LIN {X 0,Y 249.471,Z 292.033,A -85,B 0,C 180,E1 -19088.099,E2 -19088.099} C_VEL
LIN {X 0,Y 249.243,Z 292.063,A -85,B 0,C 180,E1 -19091.385,E2 -19091.385} C_VEL
LIN {X 0,Y 249.233,Z 292.064,A -85,B 0,C 180,E1 -19096.38,E2 -19096.38} C_VEL
LIN {X 0,Y 249.075,Z 292.084,A -85,B 0,C 180,E1 -19101.52,E2 -19101.52} C_VEL
LIN {X 0,Y 249.108,Z 292.08,A -85,B 0,C 180,E1 -19105.477,E2 -19105.477} C_VEL
LIN {X 0,Y 249.043,Z 292.087,A -85,B 0,C 180,E1 -19109.572,E2 -19109.572} C_VEL
LIN {X 0,Y 248.346,Z 292.177,A -85,B 0,C 180,E1 -19110.921,E2 -19110.921} C_VEL
LIN {X 0,Y 245.475,Z 292.533,A -85,B 0,C 180,E1 -19113.119,E2 -19113.119} C_VEL
LIN {X 0,Y 243.059,Z 292.835,A -85,B 0,C 180,E1 -19114.91,E2 -19114.91} C_VEL
LIN {X 0,Y 242.033,Z 292.96,A -85,B 0,C 180,E1 -19116.299,E2 -19116.299} C_VEL
LIN {X 0,Y 241.954,Z 292.965,A -85,B 0,C 180,E1 -19116.77,E2 -19116.77} C_VEL
LIN {X 0,Y 241.928,Z 292.974,A -85,B 0,C 180,E1 -19120.953,E2 -19120.953} C_VEL
LIN {X 0,Y 241.986,Z 293.122,A -85,B 0,C 180,E1 -19124.826,E2 -19124.826} C_VEL
LIN {X 0,Y 245.244,Z 306.398,A -85,B 0,C 180,E1 -19129.049,E2 -19129.049} C_VEL
LIN {X 0,Y 245.535,Z 307.451,A -85,B 0,C 180,E1 -19129.318,E2 -19129.318} C_VEL
LIN {X 0,Y 258.623,Z 343.04,A -85,B 0,C 180,E1 -19132.403,E2 -19132.403} C_VEL
LIN {X 0,Y 260.766,Z 349.359,A -85,B 0,C 180,E1 -19132.902,E2 -19132.902} C_VEL
LIN {X 0,Y 263.208,Z 370.68,A -85,B 0,C 180,E1 -19134.126,E2 -19134.126} C_VEL
LIN {X 0,Y 255.946,Z 475.253,A -85,B 0,C 180,E1 -19138.613,E2 -19138.613} C_VEL
LIN {X 0,Y 254.356,Z 491.269,A -85,B 0,C 180,E1 -19139.606,E2 -19139.606} C_VEL
LIN {X 0,Y 252.419,Z 507.536,A -85,B 0,C 180,E1 -19140.957,E2 -19140.957} C_VEL
LIN {X 0,Y 250.356,Z 523.247,A -85,B 0,C 180,E1 -19142.636,E2 -19142.636} C_VEL
LIN {X 0,Y 248.189,Z 538.255,A -85,B 0,C 180,E1 -19144.643,E2 -19144.643} C_VEL
LIN {X 0,Y 246.113,Z 551.832,A -85,B 0,C 180,E1 -19146.883,E2 -19146.883} C_VEL
LIN {X 0,Y 244.552,Z 562.301,A -85,B 0,C 180,E1 -19148.95,E2 -19148.95} C_VEL
LIN {X 0,Y 243.07,Z 573.02,A -85,B 0,C 180,E1 -19151.458,E2 -19151.458} C_VEL
LIN {X 0,Y 241.842,Z 583.648,A -85,B 0,C 180,E1 -19154.455,E2 -19154.455} C_VEL
LIN {X 0,Y 240.981,Z 592.114,A -85,B 0,C 180,E1 -19157.368,E2 -19157.368} C_VEL
LIN {X 0,Y 240.616,Z 598.213,A -85,B 0,C 180,E1 -19159.909,E2 -19159.909} C_VEL
LIN {X 0,Y 240.531,Z 603.304,A -85,B 0,C 180,E1 -19162.447,E2 -19162.447} C_VEL
LIN {X 0,Y 240.455,Z 607.393,A -85,B 0,C 180,E1 -19164.972,E2 -19164.972} C_VEL
LIN {X 0,Y 240.557,Z 611.483,A -85,B 0,C 180,E1 -19168.328,E2 -19168.328} C_VEL
LIN {X 0,Y 240.593,Z 612.96,A -85,B 0,C 180,E1 -19170.002,E2 -19170.002} C_VEL
LIN {X 0,Y 240.362,Z 614.057,A -85,B 0,C 180,E1 -19171.678,E2 -19171.678} C_VEL
LIN {X 0,Y 240.044,Z 615.345,A -85,B 0,C 180,E1 -19175.459,E2 -19175.459} C_VEL
LIN {X 0,Y 239.986,Z 615.305,A -85,B 0,C 180,E1 -19178.422,E2 -19178.422} C_VEL
LIN {X 0,Y 240.478,Z 614.105,A -85,B 0,C 180,E1 -19181.807,E2 -19181.807} C_VEL
LIN {X 0,Y 241.79,Z 611.803,A -85,B 0,C 180,E1 -19185.167,E2 -19185.167} C_VEL
LIN {X 0,Y 243.891,Z 608.419,A -85,B 0,C 180,E1 -19188.482,E2 -19188.482} C_VEL
LIN {X 0,Y 246.847,Z 603.914,A -85,B 0,C 180,E1 -19191.725,E2 -19191.725} C_VEL
LIN {X 0,Y 251.642,Z 596.638,A -85,B 0,C 180,E1 -19195.653,E2 -19195.653} C_VEL
LIN {X 0,Y 255.249,Z 591.329,A -85,B 0,C 180,E1 -19197.912,E2 -19197.912} C_VEL
LIN {X 0,Y 261.608,Z 582.045,A -85,B 0,C 180,E1 -19201.143,E2 -19201.143} C_VEL
LIN {X 0,Y 269.062,Z 570.962,A -85,B 0,C 180,E1 -19204.168,E2 -19204.168} C_VEL
LIN {X 0,Y 276.626,Z 559.345,A -85,B 0,C 180,E1 -19206.66,E2 -19206.66} C_VEL
LIN {X 0,Y 283.903,Z 547.619,A -85,B 0,C 180,E1 -19208.689,E2 -19208.689} C_VEL
LIN {X 0,Y 291.346,Z 535.032,A -85,B 0,C 180,E1 -19210.415,E2 -19210.415} C_VEL
LIN {X 0,Y 299.334,Z 520.498,A -85,B 0,C 180,E1 -19212.003,E2 -19212.003} C_VEL
LIN {X 0,Y 305.927,Z 507.36,A -85,B 0,C 180,E1 -19213.115,E2 -19213.115} C_VEL
LIN {X 0,Y 313.351,Z 490.898,A -85,B 0,C 180,E1 -19214.214,E2 -19214.214} C_VEL
LIN {X 0,Y 320.433,Z 472.33,A -85,B 0,C 180,E1 -19215.159,E2 -19215.159} C_VEL
LIN {X 0,Y 322.394,Z 466.476,A -85,B 0,C 180,E1 -19215.395,E2 -19215.395} C_VEL
LIN {X 0,Y 321.993,Z 467.661,A -85,B 0,C 180,E1 -19215.696,E2 -19215.696} C_VEL
LIN {X 0,Y 316.048,Z 483.579,A -85,B 0,C 180,E1 -19216.64,E2 -19216.64} C_VEL
LIN {X 0,Y 309.726,Z 497.956,A -85,B 0,C 180,E1 -19217.76,E2 -19217.76} C_VEL
LIN {X 0,Y 302.493,Z 512.424,A -85,B 0,C 180,E1 -19219.197,E2 -19219.197} C_VEL
LIN {X 0,Y 295.181,Z 525.593,A -85,B 0,C 180,E1 -19220.879,E2 -19220.879} C_VEL
LIN {X 0,Y 287.732,Z 537.835,A -85,B 0,C 180,E1 -19222.804,E2 -19222.804} C_VEL
LIN {X 0,Y 280.816,Z 548.308,A -85,B 0,C 180,E1 -19224.856,E2 -19224.856} C_VEL
LIN {X 0,Y 273.456,Z 558.626,A -85,B 0,C 180,E1 -19227.335,E2 -19227.335} C_VEL
LIN {X 0,Y 266.928,Z 567.216,A -85,B 0,C 180,E1 -19229.982,E2 -19229.982} C_VEL
LIN {X 0,Y 261.165,Z 574.375,A -85,B 0,C 180,E1 -19232.775,E2 -19232.775} C_VEL
LIN {X 0,Y 256.074,Z 580.239,A -85,B 0,C 180,E1 -19235.689,E2 -19235.689} C_VEL
LIN {X 0,Y 251.537,Z 584.921,A -85,B 0,C 180,E1 -19238.701,E2 -19238.701} C_VEL
LIN {X 0,Y 248.05,Z 588.36,A -85,B 0,C 180,E1 -19241.839,E2 -19241.839} C_VEL
LIN {X 0,Y 245.208,Z 590.711,A -85,B 0,C 180,E1 -19245.05,E2 -19245.05} C_VEL
LIN {X 0,Y 243.186,Z 591.965,A -85,B 0,C 180,E1 -19248.327,E2 -19248.327} C_VEL
LIN {X 0,Y 241.569,Z 592.097,A -85,B 0,C 180,E1 -19251.635,E2 -19251.635} C_VEL
LIN {X 0,Y 240.677,Z 591.061,A -85,B 0,C 180,E1 -19254.973,E2 -19254.973} C_VEL
LIN {X 0,Y 240.242,Z 588.872,A -85,B 0,C 180,E1 -19258.322,E2 -19258.322} C_VEL
LIN {X 0,Y 240.107,Z 585.46,A -85,B 0,C 180,E1 -19261.676,E2 -19261.676} C_VEL
LIN {X 0,Y 240.137,Z 580.702,A -85,B 0,C 180,E1 -19265.036,E2 -19265.036} C_VEL
LIN {X 0,Y 240.498,Z 574.473,A -85,B 0,C 180,E1 -19268.4,E2 -19268.4} C_VEL
LIN {X 0,Y 241.056,Z 567.663,A -85,B 0,C 180,E1 -19271.348,E2 -19271.348} C_VEL
LIN {X 0,Y 242.08,Z 559.425,A -85,B 0,C 180,E1 -19274.285,E2 -19274.285} C_VEL
LIN {X 0,Y 243.19,Z 549.848,A -85,B 0,C 180,E1 -19277.122,E2 -19277.122} C_VEL
LIN {X 0,Y 244.711,Z 539.338,A -85,B 0,C 180,E1 -19279.72,E2 -19279.72} C_VEL
LIN {X 0,Y 246.494,Z 527.366,A -85,B 0,C 180,E1 -19282.195,E2 -19282.195} C_VEL
LIN {X 0,Y 248.317,Z 514.289,A -85,B 0,C 180,E1 -19284.45,E2 -19284.45} C_VEL
LIN {X 0,Y 250.42,Z 499.832,A -85,B 0,C 180,E1 -19286.501,E2 -19286.501} C_VEL
LIN {X 0,Y 252.301,Z 484.557,A -85,B 0,C 180,E1 -19288.263,E2 -19288.263} C_VEL
LIN {X 0,Y 253.967,Z 469.508,A -85,B 0,C 180,E1 -19289.645,E2 -19289.645} C_VEL
LIN {X 0,Y 255.476,Z 453.024,A -85,B 0,C 180,E1 -19290.82,E2 -19290.82} C_VEL
LIN {X 0,Y 256.778,Z 434.752,A -85,B 0,C 180,E1 -19291.74,E2 -19291.74} C_VEL
LIN {X 0,Y 263.19,Z 342.406,A -85,B 0,C 180,E1 -19295.61,E2 -19295.61} C_VEL
LIN {X 0,Y 247.394,Z 305.685,A -85,B 0,C 180,E1 -19298.918,E2 -19298.918} C_VEL
LIN {X 0,Y 242.129,Z 293.792,A -85,B 0,C 180,E1 -19300.101,E2 -19300.101} C_VEL
LIN {X 0,Y 241.983,Z 292.971,A -85,B 0,C 180,E1 -19300.199,E2 -19300.199} C_VEL
LIN {X 0,Y 241.931,Z 292.976,A -85,B 0,C 180,E1 -19304.2,E2 -19304.2} C_VEL
LIN {X 0,Y 241.938,Z 292.973,A -85,B 0,C 180,E1 -19308.075,E2 -19308.075} C_VEL
LIN {X 0,Y 241.989,Z 292.966,A -85,B 0,C 180,E1 -19312.416,E2 -19312.416} C_VEL
LIN {X 0,Y 241.978,Z 292.968,A -85,B 0,C 180,E1 -19316.505,E2 -19316.505} C_VEL
LIN {X 0,Y 241.975,Z 292.966,A -85,B 0,C 180,E1 -19320.61,E2 -19320.61} C_VEL
LIN {X 0,Y 242.03,Z 292.961,A -85,B 0,C 180,E1 -19324.176,E2 -19324.176} C_VEL
LIN {X 0,Y 242.019,Z 292.963,A -85,B 0,C 180,E1 -19328.313,E2 -19328.313} C_VEL
LIN {X 0,Y 242.111,Z 292.952,A -85,B 0,C 180,E1 -19333.314,E2 -19333.314} C_VEL
LIN {X 0,Y 242.178,Z 292.943,A -85,B 0,C 180,E1 -19338.277,E2 -19338.277} C_VEL
LIN {X 0,Y 242.422,Z 292.915,A -85,B 0,C 180,E1 -19341.663,E2 -19341.663} C_VEL
LIN {X 0,Y 242.251,Z 292.932,A -85,B 0,C 180,E1 -19345.005,E2 -19345.005} C_VEL
LIN {X 0,Y 242.629,Z 292.885,A -85,B 0,C 180,E1 -19348.338,E2 -19348.338} C_VEL
LIN {X 0,Y 242.629,Z 292.886,A -85,B 0,C 180,E1 -19351.658,E2 -19351.658} C_VEL
LIN {X 0,Y 242.425,Z 292.91,A -85,B 0,C 180,E1 -19356.657,E2 -19356.657} C_VEL
LIN {X 0,Y 242.306,Z 292.924,A -85,B 0,C 180,E1 -19360.02,E2 -19360.02} C_VEL
LIN {X 0,Y 242.157,Z 292.946,A -85,B 0,C 180,E1 -19365.139,E2 -19365.139} C_VEL
LIN {X 0,Y 242.063,Z 292.953,A -85,B 0,C 180,E1 -19368.622,E2 -19368.622} C_VEL
LIN {X 0,Y 242.003,Z 292.963,A -85,B 0,C 180,E1 -19372.178,E2 -19372.178} C_VEL
LIN {X 0,Y 242.056,Z 292.956,A -85,B 0,C 180,E1 -19375.836,E2 -19375.836} C_VEL
LIN {X 0,Y 241.996,Z 292.966,A -85,B 0,C 180,E1 -19379.582,E2 -19379.582} C_VEL
LIN {X 0,Y 241.979,Z 292.968,A -85,B 0,C 180,E1 -19383.49,E2 -19383.49} C_VEL
LIN {X 0,Y 241.987,Z 292.967,A -85,B 0,C 180,E1 -19387.579,E2 -19387.579} C_VEL
LIN {X 0,Y 241.926,Z 292.972,A -85,B 0,C 180,E1 -19391.921,E2 -19391.921} C_VEL
LIN {X 0,Y 241.924,Z 292.973,A -85,B 0,C 180,E1 -19396.57,E2 -19396.57} C_VEL
LIN {X 0,Y 241.943,Z 292.97,A -85,B 0,C 180,E1 -19400.28,E2 -19400.28} C_VEL
LIN {X 0,Y 241.974,Z 292.966,A -85,B 0,C 180,E1 -19404.489,E2 -19404.489} C_VEL
LIN {X 0,Y 241.962,Z 292.968,A -85,B 0,C 180,E1 -19408.48,E2 -19408.48} C_VEL
LIN {X 0,Y 241.994,Z 292.963,A -85,B 0,C 180,E1 -19412.313,E2 -19412.313} C_VEL
LIN {X 0,Y 242.028,Z 292.96,A -85,B 0,C 180,E1 -19416.015,E2 -19416.015} C_VEL
LIN {X 0,Y 242.022,Z 292.96,A -85,B 0,C 180,E1 -19419.608,E2 -19419.608} C_VEL
LIN {X 0,Y 242.151,Z 292.948,A -85,B 0,C 180,E1 -19423.279,E2 -19423.279} C_VEL
LIN {X 0,Y 242.174,Z 292.939,A -85,B 0,C 180,E1 -19428.281,E2 -19428.281} C_VEL
LIN {X 0,Y 242.414,Z 292.912,A -85,B 0,C 180,E1 -19431.667,E2 -19431.667} C_VEL
LIN {X 0,Y 242.246,Z 292.936,A -85,B 0,C 180,E1 -19435.008,E2 -19435.008} C_VEL
LIN {X 0,Y 242.625,Z 292.885,A -85,B 0,C 180,E1 -19438.341,E2 -19438.341} C_VEL
LIN {X 0,Y 242.625,Z 292.885,A -85,B 0,C 180,E1 -19441.661,E2 -19441.661} C_VEL
LIN {X 0,Y 242.422,Z 292.912,A -85,B 0,C 180,E1 -19446.66,E2 -19446.66} C_VEL
LIN {X 0,Y 242.304,Z 292.925,A -85,B 0,C 180,E1 -19450.023,E2 -19450.023} C_VEL
LIN {X 0,Y 242.157,Z 292.947,A -85,B 0,C 180,E1 -19455.143,E2 -19455.143} C_VEL
LIN {X 0,Y 242.062,Z 292.959,A -85,B 0,C 180,E1 -19458.626,E2 -19458.626} C_VEL
LIN {X 0,Y 241.997,Z 292.966,A -85,B 0,C 180,E1 -19462.183,E2 -19462.183} C_VEL
LIN {X 0,Y 242.059,Z 292.958,A -85,B 0,C 180,E1 -19465.84,E2 -19465.84} C_VEL
LIN {X 0,Y 242.023,Z 292.962,A -85,B 0,C 180,E1 -19469.582,E2 -19469.582} C_VEL
LIN {X 0,Y 241.973,Z 292.968,A -85,B 0,C 180,E1 -19473.495,E2 -19473.495} C_VEL
LIN {X 0,Y 241.954,Z 292.965,A -85,B 0,C 180,E1 -19476.77,E2 -19476.77} C_VEL
LIN {X 0,Y 241.262,Z 293.057,A -85,B 0,C 180,E1 -19478.16,E2 -19478.16} C_VEL
LIN {X 0,Y 238.301,Z 293.425,A -85,B 0,C 180,E1 -19480.425,E2 -19480.425} C_VEL
LIN {X 0,Y 235.86,Z 293.727,A -85,B 0,C 180,E1 -19482.272,E2 -19482.272} C_VEL
LIN {X 0,Y 234.923,Z 293.843,A -85,B 0,C 180,E1 -19483.708,E2 -19483.708} C_VEL
LIN {X 0,Y 234.906,Z 293.846,A -85,B 0,C 180,E1 -19484.193,E2 -19484.193} C_VEL
LIN {X 0,Y 238.061,Z 306.82,A -85,B 0,C 180,E1 -19488.475,E2 -19488.475} C_VEL
LIN {X 0,Y 251.779,Z 344.086,A -85,B 0,C 180,E1 -19491.829,E2 -19491.829} C_VEL
LIN {X 0,Y 254.286,Z 351.542,A -85,B 0,C 180,E1 -19492.432,E2 -19492.432} C_VEL
LIN {X 0,Y 256.465,Z 371.959,A -85,B 0,C 180,E1 -19493.631,E2 -19493.631} C_VEL
LIN {X 0,Y 249.049,Z 475.308,A -85,B 0,C 180,E1 -19498.236,E2 -19498.236} C_VEL
LIN {X 0,Y 247.449,Z 491.177,A -85,B 0,C 180,E1 -19499.257,E2 -19499.257} C_VEL
LIN {X 0,Y 245.48,Z 507.314,A -85,B 0,C 180,E1 -19500.644,E2 -19500.644} C_VEL
LIN {X 0,Y 243.495,Z 522.086,A -85,B 0,C 180,E1 -19502.266,E2 -19502.266} C_VEL
LIN {X 0,Y 241.306,Z 536.878,A -85,B 0,C 180,E1 -19504.283,E2 -19504.283} C_VEL
LIN {X 0,Y 239.163,Z 550.864,A -85,B 0,C 180,E1 -19506.63,E2 -19506.63} C_VEL
LIN {X 0,Y 237.259,Z 563.298,A -85,B 0,C 180,E1 -19509.181,E2 -19509.181} C_VEL
LIN {X 0,Y 235.803,Z 573.803,A -85,B 0,C 180,E1 -19511.766,E2 -19511.766} C_VEL
LIN {X 0,Y 234.669,Z 584.034,A -85,B 0,C 180,E1 -19514.811,E2 -19514.811} C_VEL
LIN {X 0,Y 233.873,Z 592.449,A -85,B 0,C 180,E1 -19517.859,E2 -19517.859} C_VEL
LIN {X 0,Y 233.529,Z 598.435,A -85,B 0,C 180,E1 -19520.475,E2 -19520.475} C_VEL
LIN {X 0,Y 233.493,Z 603.825,A -85,B 0,C 180,E1 -19523.361,E2 -19523.361} C_VEL
LIN {X 0,Y 233.399,Z 608.437,A -85,B 0,C 180,E1 -19526.55,E2 -19526.55} C_VEL
LIN {X 0,Y 233.51,Z 610.412,A -85,B 0,C 180,E1 -19528.278,E2 -19528.278} C_VEL
LIN {X 0,Y 233.579,Z 612.003,A -85,B 0,C 180,E1 -19530.002,E2 -19530.002} C_VEL
LIN {X 0,Y 233.316,Z 613.2,A -85,B 0,C 180,E1 -19531.728,E2 -19531.728} C_VEL
LIN {X 0,Y 232.98,Z 614.68,A -85,B 0,C 180,E1 -19535.449,E2 -19535.449} C_VEL
LIN {X 0,Y 232.934,Z 614.788,A -85,B 0,C 180,E1 -19538.679,E2 -19538.679} C_VEL
LIN {X 0,Y 233.467,Z 613.824,A -85,B 0,C 180,E1 -19542.167,E2 -19542.167} C_VEL
LIN {X 0,Y 234.887,Z 611.793,A -85,B 0,C 180,E1 -19545.624,E2 -19545.624} C_VEL
LIN {X 0,Y 237.113,Z 608.634,A -85,B 0,C 180,E1 -19549.031,E2 -19549.031} C_VEL
LIN {X 0,Y 240.255,Z 604.391,A -85,B 0,C 180,E1 -19552.353,E2 -19552.353} C_VEL
LIN {X 0,Y 244.203,Z 599.074,A -85,B 0,C 180,E1 -19555.577,E2 -19555.577} C_VEL
LIN {X 0,Y 247.692,Z 594.319,A -85,B 0,C 180,E1 -19557.918,E2 -19557.918} C_VEL
LIN {X 0,Y 254.219,Z 585.86,A -85,B 0,C 180,E1 -19561.223,E2 -19561.223} C_VEL
LIN {X 0,Y 261.679,Z 575.783,A -85,B 0,C 180,E1 -19564.335,E2 -19564.335} C_VEL
LIN {X 0,Y 269.264,Z 565.268,A -85,B 0,C 180,E1 -19566.895,E2 -19566.895} C_VEL
LIN {X 0,Y 277.722,Z 553.047,A -85,B 0,C 180,E1 -19569.248,E2 -19569.248} C_VEL
LIN {X 0,Y 285.828,Z 540.646,A -85,B 0,C 180,E1 -19571.129,E2 -19571.129} C_VEL
LIN {X 0,Y 294.614,Z 526.272,A -85,B 0,C 180,E1 -19572.835,E2 -19572.835} C_VEL
LIN {X 0,Y 301.989,Z 513.063,A -85,B 0,C 180,E1 -19574.05,E2 -19574.05} C_VEL
LIN {X 0,Y 310.398,Z 496.278,A -85,B 0,C 180,E1 -19575.244,E2 -19575.244} C_VEL
LIN {X 0,Y 311.954,Z 492.865,A -85,B 0,C 180,E1 -19575.438,E2 -19575.438} C_VEL
LIN {X 0,Y 312.63,Z 491.313,A -85,B 0,C 180,E1 -19575.821,E2 -19575.821} C_VEL
LIN {X 0,Y 304.858,Z 506.763,A -85,B 0,C 180,E1 -19577.15,E2 -19577.15} C_VEL
LIN {X 0,Y 297.467,Z 519.809,A -85,B 0,C 180,E1 -19578.582,E2 -19578.582} C_VEL
LIN {X 0,Y 289.388,Z 532.714,A -85,B 0,C 180,E1 -19580.393,E2 -19580.393} C_VEL
LIN {X 0,Y 281.786,Z 543.831,A -85,B 0,C 180,E1 -19582.333,E2 -19582.333} C_VEL
LIN {X 0,Y 273.714,Z 554.743,A -85,B 0,C 180,E1 -19584.709,E2 -19584.709} C_VEL
LIN {X 0,Y 266.275,Z 563.98,A -85,B 0,C 180,E1 -19587.242,E2 -19587.242} C_VEL
LIN {X 0,Y 259.516,Z 571.879,A -85,B 0,C 180,E1 -19590.022,E2 -19590.022} C_VEL
LIN {X 0,Y 253.824,Z 578.109,A -85,B 0,C 180,E1 -19592.814,E2 -19592.814} C_VEL
LIN {X 0,Y 248.587,Z 583.315,A -85,B 0,C 180,E1 -19595.798,E2 -19595.798} C_VEL
LIN {X 0,Y 245.121,Z 586.469,A -85,B 0,C 180,E1 -19598.115,E2 -19598.115} C_VEL
LIN {X 0,Y 241.423,Z 589.63,A -85,B 0,C 180,E1 -19601.323,E2 -19601.323} C_VEL
LIN {X 0,Y 238.419,Z 591.673,A -85,B 0,C 180,E1 -19604.614,E2 -19604.614} C_VEL
LIN {X 0,Y 236.267,Z 592.64,A -85,B 0,C 180,E1 -19607.981,E2 -19607.981} C_VEL
LIN {X 0,Y 234.5,Z 592.517,A -85,B 0,C 180,E1 -19611.51,E2 -19611.51} C_VEL
LIN {X 0,Y 233.615,Z 591.322,A -85,B 0,C 180,E1 -19614.821,E2 -19614.821} C_VEL
LIN {X 0,Y 233.169,Z 588.895,A -85,B 0,C 180,E1 -19618.271,E2 -19618.271} C_VEL
LIN {X 0,Y 233.012,Z 585.241,A -85,B 0,C 180,E1 -19621.727,E2 -19621.727} C_VEL
LIN {X 0,Y 233.063,Z 580.242,A -85,B 0,C 180,E1 -19625.189,E2 -19625.189} C_VEL
LIN {X 0,Y 233.457,Z 573.753,A -85,B 0,C 180,E1 -19628.656,E2 -19628.656} C_VEL
LIN {X 0,Y 234.039,Z 566.675,A -85,B 0,C 180,E1 -19631.693,E2 -19631.693} C_VEL
LIN {X 0,Y 235.137,Z 558.152,A -85,B 0,C 180,E1 -19634.716,E2 -19634.716} C_VEL
LIN {X 0,Y 236.389,Z 547.893,A -85,B 0,C 180,E1 -19637.726,E2 -19637.726} C_VEL
LIN {X 0,Y 237.919,Z 537.359,A -85,B 0,C 180,E1 -19640.308,E2 -19640.308} C_VEL
LIN {X 0,Y 239.844,Z 524.995,A -85,B 0,C 180,E1 -19642.844,E2 -19642.844} C_VEL
LIN {X 0,Y 241.761,Z 511.435,A -85,B 0,C 180,E1 -19645.158,E2 -19645.158} C_VEL
LIN {X 0,Y 243.852,Z 496.676,A -85,B 0,C 180,E1 -19647.218,E2 -19647.218} C_VEL
LIN {X 0,Y 245.794,Z 481.08,A -85,B 0,C 180,E1 -19648.965,E2 -19648.965} C_VEL
LIN {X 0,Y 247.553,Z 465.099,A -85,B 0,C 180,E1 -19650.376,E2 -19650.376} C_VEL
LIN {X 0,Y 248.997,Z 447.809,A -85,B 0,C 180,E1 -19651.535,E2 -19651.535} C_VEL
LIN {X 0,Y 251.431,Z 412.603,A -85,B 0,C 180,E1 -19653.162,E2 -19653.162} C_VEL
LIN {X 0,Y 256.429,Z 344.058,A -85,B 0,C 180,E1 -19656.119,E2 -19656.119} C_VEL
LIN {X 0,Y 241.327,Z 308.785,A -85,B 0,C 180,E1 -19659.384,E2 -19659.384} C_VEL
LIN {X 0,Y 234.952,Z 294.19,A -85,B 0,C 180,E1 -19660.864,E2 -19660.864} C_VEL
LIN {X 0,Y 234.911,Z 293.85,A -85,B 0,C 180,E1 -19660.918,E2 -19660.918} C_VEL
LIN {X 0,Y 234.895,Z 293.853,A -85,B 0,C 180,E1 -19664.102,E2 -19664.102} C_VEL
LIN {X 0,Y 234.883,Z 293.85,A -85,B 0,C 180,E1 -19668.83,E2 -19668.83} C_VEL
LIN {X 0,Y 234.918,Z 293.845,A -85,B 0,C 180,E1 -19671.076,E2 -19671.076} C_VEL
LIN {X 0,Y 234.929,Z 293.845,A -85,B 0,C 180,E1 -19675.359,E2 -19675.359} C_VEL
LIN {X 0,Y 234.897,Z 293.848,A -85,B 0,C 180,E1 -19679.425,E2 -19679.425} C_VEL
LIN {X 0,Y 234.966,Z 293.843,A -85,B 0,C 180,E1 -19683.804,E2 -19683.804} C_VEL
LIN {X 0,Y 234.965,Z 293.841,A -85,B 0,C 180,E1 -19688.963,E2 -19688.963} C_VEL
LIN {X 0,Y 235.052,Z 293.831,A -85,B 0,C 180,E1 -19693.09,E2 -19693.09} C_VEL
LIN {X 0,Y 235.108,Z 293.825,A -85,B 0,C 180,E1 -19697.919,E2 -19697.919} C_VEL
LIN {X 0,Y 235.372,Z 293.794,A -85,B 0,C 180,E1 -19701.412,E2 -19701.412} C_VEL
LIN {X 0,Y 235.398,Z 293.787,A -85,B 0,C 180,E1 -19703.139,E2 -19703.139} C_VEL
LIN {X 0,Y 235.588,Z 293.763,A -85,B 0,C 180,E1 -19708.288,E2 -19708.288} C_VEL
LIN {X 0,Y 235.588,Z 293.763,A -85,B 0,C 180,E1 -19711.707,E2 -19711.707} C_VEL
LIN {X 0,Y 235.396,Z 293.786,A -85,B 0,C 180,E1 -19716.856,E2 -19716.856} C_VEL
LIN {X 0,Y 235.23,Z 293.804,A -85,B 0,C 180,E1 -19720.324,E2 -19720.324} C_VEL
LIN {X 0,Y 235.104,Z 293.825,A -85,B 0,C 180,E1 -19725.604,E2 -19725.604} C_VEL
LIN {X 0,Y 234.999,Z 293.835,A -85,B 0,C 180,E1 -19729.204,E2 -19729.204} C_VEL
LIN {X 0,Y 234.951,Z 293.842,A -85,B 0,C 180,E1 -19732.881,E2 -19732.881} C_VEL
LIN {X 0,Y 234.957,Z 293.839,A -85,B 0,C 180,E1 -19736.656,E2 -19736.656} C_VEL
LIN {X 0,Y 234.911,Z 293.846,A -85,B 0,C 180,E1 -19740.568,E2 -19740.568} C_VEL
LIN {X 0,Y 234.949,Z 293.84,A -85,B 0,C 180,E1 -19744.632,E2 -19744.632} C_VEL
LIN {X 0,Y 234.93,Z 293.845,A -85,B 0,C 180,E1 -19748.943,E2 -19748.943} C_VEL
LIN {X 0,Y 234.877,Z 293.851,A -85,B 0,C 180,E1 -19753.485,E2 -19753.485} C_VEL
LIN {X 0,Y 234.877,Z 293.85,A -85,B 0,C 180,E1 -19756.514,E2 -19756.514} C_VEL
LIN {X 0,Y 234.905,Z 293.849,A -85,B 0,C 180,E1 -19761.078,E2 -19761.078} C_VEL
LIN {X 0,Y 234.917,Z 293.849,A -85,B 0,C 180,E1 -19765.362,E2 -19765.362} C_VEL
LIN {X 0,Y 234.919,Z 293.846,A -85,B 0,C 180,E1 -19769.432,E2 -19769.432} C_VEL
LIN {X 0,Y 234.981,Z 293.838,A -85,B 0,C 180,E1 -19773.794,E2 -19773.794} C_VEL
LIN {X 0,Y 234.985,Z 293.838,A -85,B 0,C 180,E1 -19778.969,E2 -19778.969} C_VEL
LIN {X 0,Y 235.084,Z 293.828,A -85,B 0,C 180,E1 -19783.06,E2 -19783.06} C_VEL
LIN {X 0,Y 235.134,Z 293.816,A -85,B 0,C 180,E1 -19787.925,E2 -19787.925} C_VEL
LIN {X 0,Y 235.364,Z 293.792,A -85,B 0,C 180,E1 -19791.415,E2 -19791.415} C_VEL
LIN {X 0,Y 235.39,Z 293.79,A -85,B 0,C 180,E1 -19793.142,E2 -19793.142} C_VEL
LIN {X 0,Y 235.584,Z 293.762,A -85,B 0,C 180,E1 -19798.292,E2 -19798.292} C_VEL
LIN {X 0,Y 235.584,Z 293.762,A -85,B 0,C 180,E1 -19801.711,E2 -19801.711} C_VEL
LIN {X 0,Y 235.393,Z 293.789,A -85,B 0,C 180,E1 -19806.86,E2 -19806.86} C_VEL
LIN {X 0,Y 235.228,Z 293.807,A -85,B 0,C 180,E1 -19810.328,E2 -19810.328} C_VEL
LIN {X 0,Y 235.104,Z 293.823,A -85,B 0,C 180,E1 -19815.608,E2 -19815.608} C_VEL
LIN {X 0,Y 234.998,Z 293.84,A -85,B 0,C 180,E1 -19819.208,E2 -19819.208} C_VEL
LIN {X 0,Y 234.944,Z 293.849,A -85,B 0,C 180,E1 -19822.886,E2 -19822.886} C_VEL
LIN {X 0,Y 234.961,Z 293.845,A -85,B 0,C 180,E1 -19826.66,E2 -19826.66} C_VEL
LIN {X 0,Y 234.924,Z 293.848,A -85,B 0,C 180,E1 -19830.57,E2 -19830.57} C_VEL
LIN {X 0,Y 234.923,Z 293.848,A -85,B 0,C 180,E1 -19834.64,E2 -19834.64} C_VEL
LIN {X 0,Y 234.936,Z 293.845,A -85,B 0,C 180,E1 -19838.947,E2 -19838.947} C_VEL
LIN {X 0,Y 234.885,Z 293.848,A -85,B 0,C 180,E1 -19843.488,E2 -19843.488} C_VEL
LIN {X 0,Y 234.906,Z 293.846,A -85,B 0,C 180,E1 -19844.193,E2 -19844.193} C_VEL
LIN {X 0,Y 234.529,Z 297.073,A -85,B 0,C 180,E1 -19845.175,E2 -19845.175} C_VEL
LIN {X 0,Y 231.193,Z 305.933,A -85,B 0,C 180,E1 -19847.406,E2 -19847.406} C_VEL
LIN {X 0,Y 231.341,Z 308.208,A -85,B 0,C 180,E1 -19847.796,E2 -19847.796} C_VEL
LIN {X 0,Y 231.483,Z 308.699,A -85,B 0,C 180,E1 -19847.849,E2 -19847.849} C_VEL
LIN {X 0,Y 244.35,Z 343.383,A -85,B 0,C 180,E1 -19851.089,E2 -19851.089} C_VEL
LIN {X 0,Y 247.822,Z 353.873,A -85,B 0,C 180,E1 -19851.962,E2 -19851.962} C_VEL
LIN {X 0,Y 249.807,Z 372.241,A -85,B 0,C 180,E1 -19853.084,E2 -19853.084} C_VEL
LIN {X 0,Y 242.249,Z 474.246,A -85,B 0,C 180,E1 -19857.789,E2 -19857.789} C_VEL
LIN {X 0,Y 240.547,Z 490.797,A -85,B 0,C 180,E1 -19858.887,E2 -19858.887} C_VEL
LIN {X 0,Y 238.54,Z 506.868,A -85,B 0,C 180,E1 -19860.311,E2 -19860.311} C_VEL
LIN {X 0,Y 236.421,Z 522.486,A -85,B 0,C 180,E1 -19862.086,E2 -19862.086} C_VEL
LIN {X 0,Y 234.338,Z 536.071,A -85,B 0,C 180,E1 -19864.004,E2 -19864.004} C_VEL
LIN {X 0,Y 232.207,Z 549.77,A -85,B 0,C 180,E1 -19866.361,E2 -19866.361} C_VEL
LIN {X 0,Y 230.258,Z 562.314,A -85,B 0,C 180,E1 -19868.986,E2 -19868.986} C_VEL
LIN {X 0,Y 228.788,Z 572.89,A -85,B 0,C 180,E1 -19871.65,E2 -19871.65} C_VEL
LIN {X 0,Y 227.621,Z 583.202,A -85,B 0,C 180,E1 -19874.788,E2 -19874.788} C_VEL
LIN {X 0,Y 226.832,Z 591.666,A -85,B 0,C 180,E1 -19877.931,E2 -19877.931} C_VEL
LIN {X 0,Y 226.477,Z 598.592,A -85,B 0,C 180,E1 -19881.077,E2 -19881.077} C_VEL
LIN {X 0,Y 226.458,Z 603.746,A -85,B 0,C 180,E1 -19883.998,E2 -19883.998} C_VEL
LIN {X 0,Y 226.409,Z 608.273,A -85,B 0,C 180,E1 -19887.334,E2 -19887.334} C_VEL
LIN {X 0,Y 226.563,Z 611.006,A -85,B 0,C 180,E1 -19890.002,E2 -19890.002} C_VEL
LIN {X 0,Y 225.974,Z 613.212,A -85,B 0,C 180,E1 -19893.569,E2 -19893.569} C_VEL
LIN {X 0,Y 225.935,Z 613.901,A -85,B 0,C 180,E1 -19895.488,E2 -19895.488} C_VEL
LIN {X 0,Y 225.871,Z 614.253,A -85,B 0,C 180,E1 -19898.953,E2 -19898.953} C_VEL
LIN {X 0,Y 226.468,Z 613.546,A -85,B 0,C 180,E1 -19902.549,E2 -19902.549} C_VEL
LIN {X 0,Y 228.002,Z 611.698,A -85,B 0,C 180,E1 -19906.109,E2 -19906.109} C_VEL
LIN {X 0,Y 230.366,Z 608.818,A -85,B 0,C 180,E1 -19909.611,E2 -19909.611} C_VEL
LIN {X 0,Y 233.708,Z 604.914,A -85,B 0,C 180,E1 -19913.015,E2 -19913.015} C_VEL
LIN {X 0,Y 239.022,Z 598.488,A -85,B 0,C 180,E1 -19917.115,E2 -19917.115} C_VEL
LIN {X 0,Y 242.996,Z 593.772,A -85,B 0,C 180,E1 -19919.453,E2 -19919.453} C_VEL
LIN {X 0,Y 249.94,Z 585.498,A -85,B 0,C 180,E1 -19922.773,E2 -19922.773} C_VEL
LIN {X 0,Y 257.979,Z 575.635,A -85,B 0,C 180,E1 -19925.856,E2 -19925.856} C_VEL
LIN {X 0,Y 266.026,Z 565.377,A -85,B 0,C 180,E1 -19928.379,E2 -19928.379} C_VEL
LIN {X 0,Y 274.94,Z 553.485,A -85,B 0,C 180,E1 -19930.682,E2 -19930.682} C_VEL
LIN {X 0,Y 283.489,Z 541.455,A -85,B 0,C 180,E1 -19932.499,E2 -19932.499} C_VEL
LIN {X 0,Y 291.95,Z 528.629,A -85,B 0,C 180,E1 -19934.037,E2 -19934.037} C_VEL
LIN {X 0,Y 299.4,Z 516.422,A -85,B 0,C 180,E1 -19935.195,E2 -19935.195} C_VEL
LIN {X 0,Y 303.894,Z 508.474,A -85,B 0,C 180,E1 -19935.803,E2 -19935.803} C_VEL
LIN {X 0,Y 295.567,Z 522.09,A -85,B 0,C 180,E1 -19937.337,E2 -19937.337} C_VEL
LIN {X 0,Y 287.102,Z 534.606,A -85,B 0,C 180,E1 -19939.093,E2 -19939.093} C_VEL
LIN {X 0,Y 279.089,Z 545.405,A -85,B 0,C 180,E1 -19940.982,E2 -19940.982} C_VEL
LIN {X 0,Y 270.55,Z 555.988,A -85,B 0,C 180,E1 -19943.311,E2 -19943.311} C_VEL
LIN {X 0,Y 262.644,Z 565.032,A -85,B 0,C 180,E1 -19945.809,E2 -19945.809} C_VEL
LIN {X 0,Y 255.577,Z 572.597,A -85,B 0,C 180,E1 -19948.501,E2 -19948.501} C_VEL
LIN {X 0,Y 249.254,Z 578.89,A -85,B 0,C 180,E1 -19951.357,E2 -19951.357} C_VEL
LIN {X 0,Y 243.675,Z 583.972,A -85,B 0,C 180,E1 -19954.365,E2 -19954.365} C_VEL
LIN {X 0,Y 238.721,Z 587.964,A -85,B 0,C 180,E1 -19957.496,E2 -19957.496} C_VEL
LIN {X 0,Y 234.814,Z 590.811,A -85,B 0,C 180,E1 -19960.777,E2 -19960.777} C_VEL
LIN {X 0,Y 231.648,Z 592.625,A -85,B 0,C 180,E1 -19964.153,E2 -19964.153} C_VEL
LIN {X 0,Y 229.351,Z 593.32,A -85,B 0,C 180,E1 -19967.612,E2 -19967.612} C_VEL
LIN {X 0,Y 227.43,Z 592.862,A -85,B 0,C 180,E1 -19971.45,E2 -19971.45} C_VEL
LIN {X 0,Y 226.537,Z 591.465,A -85,B 0,C 180,E1 -19974.658,E2 -19974.658} C_VEL
LIN {X 0,Y 226.099,Z 588.842,A -85,B 0,C 180,E1 -19978.217,E2 -19978.217} C_VEL
LIN {X 0,Y 225.92,Z 584.978,A -85,B 0,C 180,E1 -19981.781,E2 -19981.781} C_VEL
LIN {X 0,Y 225.997,Z 579.742,A -85,B 0,C 180,E1 -19985.352,E2 -19985.352} C_VEL
LIN {X 0,Y 226.411,Z 572.977,A -85,B 0,C 180,E1 -19988.927,E2 -19988.927} C_VEL
LIN {X 0,Y 227.023,Z 565.633,A -85,B 0,C 180,E1 -19992.06,E2 -19992.06} C_VEL
LIN {X 0,Y 228.177,Z 556.791,A -85,B 0,C 180,E1 -19995.176,E2 -19995.176} C_VEL
LIN {X 0,Y 229.442,Z 546.978,A -85,B 0,C 180,E1 -19998.06,E2 -19998.06} C_VEL
LIN {X 0,Y 231.155,Z 535.304,A -85,B 0,C 180,E1 -20000.929,E2 -20000.929} C_VEL
LIN {X 0,Y 233.145,Z 522.427,A -85,B 0,C 180,E1 -20003.54,E2 -20003.54} C_VEL
LIN {X 0,Y 235.208,Z 508.234,A -85,B 0,C 180,E1 -20005.911,E2 -20005.911} C_VEL
LIN {X 0,Y 237.174,Z 494.344,A -85,B 0,C 180,E1 -20007.819,E2 -20007.819} C_VEL
LIN {X 0,Y 239.205,Z 478.306,A -85,B 0,C 180,E1 -20009.599,E2 -20009.599} C_VEL
LIN {X 0,Y 240.998,Z 461.613,A -85,B 0,C 180,E1 -20011.049,E2 -20011.049} C_VEL
LIN {X 0,Y 242.393,Z 444.81,A -85,B 0,C 180,E1 -20012.129,E2 -20012.129} C_VEL
LIN {X 0,Y 249.659,Z 345.549,A -85,B 0,C 180,E1 -20016.652,E2 -20016.652} C_VEL
LIN {X 0,Y 234.565,Z 310.363,A -85,B 0,C 180,E1 -20020.01,E2 -20020.01} C_VEL
LIN {X 0,Y 227.938,Z 295.232,A -85,B 0,C 180,E1 -20021.619,E2 -20021.619} C_VEL
LIN {X 0,Y 227.849,Z 294.73,A -85,B 0,C 180,E1 -20021.712,E2 -20021.712} C_VEL
LIN {X 0,Y 227.834,Z 294.731,A -85,B 0,C 180,E1 -20025.19,E2 -20025.19} C_VEL
LIN {X 0,Y 227.826,Z 294.732,A -85,B 0,C 180,E1 -20029.621,E2 -20029.621} C_VEL
LIN {X 0,Y 227.88,Z 294.723,A -85,B 0,C 180,E1 -20034.126,E2 -20034.126} C_VEL
LIN {X 0,Y 227.854,Z 294.725,A -85,B 0,C 180,E1 -20038.373,E2 -20038.373} C_VEL
LIN {X 0,Y 227.853,Z 294.726,A -85,B 0,C 180,E1 -20042.438,E2 -20042.438} C_VEL
LIN {X 0,Y 227.891,Z 294.721,A -85,B 0,C 180,E1 -20046.362,E2 -20046.362} C_VEL
LIN {X 0,Y 227.91,Z 294.721,A -85,B 0,C 180,E1 -20050.169,E2 -20050.169} C_VEL
LIN {X 0,Y 228.016,Z 294.71,A -85,B 0,C 180,E1 -20053.892,E2 -20053.892} C_VEL
LIN {X 0,Y 228.063,Z 294.703,A -85,B 0,C 180,E1 -20057.54,E2 -20057.54} C_VEL
LIN {X 0,Y 228.301,Z 294.673,A -85,B 0,C 180,E1 -20061.144,E2 -20061.144} C_VEL
LIN {X 0,Y 228.349,Z 294.665,A -85,B 0,C 180,E1 -20062.926,E2 -20062.926} C_VEL
LIN {X 0,Y 228.547,Z 294.64,A -85,B 0,C 180,E1 -20068.235,E2 -20068.235} C_VEL
LIN {X 0,Y 228.547,Z 294.64,A -85,B 0,C 180,E1 -20071.76,E2 -20071.76} C_VEL
LIN {X 0,Y 228.347,Z 294.665,A -85,B 0,C 180,E1 -20077.069,E2 -20077.069} C_VEL
LIN {X 0,Y 228.151,Z 294.686,A -85,B 0,C 180,E1 -20080.648,E2 -20080.648} C_VEL
LIN {X 0,Y 228.056,Z 294.701,A -85,B 0,C 180,E1 -20084.27,E2 -20084.27} C_VEL
LIN {X 0,Y 227.994,Z 294.706,A -85,B 0,C 180,E1 -20087.951,E2 -20087.951} C_VEL
LIN {X 0,Y 227.92,Z 294.717,A -85,B 0,C 180,E1 -20092.327,E2 -20092.327} C_VEL
LIN {X 0,Y 227.931,Z 294.714,A -85,B 0,C 180,E1 -20096.601,E2 -20096.601} C_VEL
LIN {X 0,Y 227.886,Z 294.721,A -85,B 0,C 180,E1 -20100.29,E2 -20100.29} C_VEL
LIN {X 0,Y 227.878,Z 294.722,A -85,B 0,C 180,E1 -20103.717,E2 -20103.717} C_VEL
LIN {X 0,Y 227.837,Z 294.727,A -85,B 0,C 180,E1 -20108.089,E2 -20108.089} C_VEL
LIN {X 0,Y 227.8,Z 294.732,A -85,B 0,C 180,E1 -20112.741,E2 -20112.741} C_VEL
LIN {X 0,Y 227.8,Z 294.736,A -85,B 0,C 180,E1 -20117.257,E2 -20117.257} C_VEL
LIN {X 0,Y 227.831,Z 294.725,A -85,B 0,C 180,E1 -20121.909,E2 -20121.909} C_VEL
LIN {X 0,Y 227.866,Z 294.724,A -85,B 0,C 180,E1 -20126.377,E2 -20126.377} C_VEL
LIN {X 0,Y 227.906,Z 294.717,A -85,B 0,C 180,E1 -20130.438,E2 -20130.438} C_VEL
LIN {X 0,Y 227.912,Z 294.718,A -85,B 0,C 180,E1 -20134.426,E2 -20134.426} C_VEL
LIN {X 0,Y 227.935,Z 294.714,A -85,B 0,C 180,E1 -20138.286,E2 -20138.286} C_VEL
LIN {X 0,Y 228.022,Z 294.706,A -85,B 0,C 180,E1 -20142.827,E2 -20142.827} C_VEL
LIN {X 0,Y 228.082,Z 294.696,A -85,B 0,C 180,E1 -20147.545,E2 -20147.545} C_VEL
LIN {X 0,Y 228.293,Z 294.674,A -85,B 0,C 180,E1 -20151.147,E2 -20151.147} C_VEL
LIN {X 0,Y 228.341,Z 294.668,A -85,B 0,C 180,E1 -20152.93,E2 -20152.93} C_VEL
LIN {X 0,Y 228.543,Z 294.639,A -85,B 0,C 180,E1 -20158.239,E2 -20158.239} C_VEL
LIN {X 0,Y 228.543,Z 294.639,A -85,B 0,C 180,E1 -20161.764,E2 -20161.764} C_VEL
LIN {X 0,Y 228.344,Z 294.668,A -85,B 0,C 180,E1 -20167.073,E2 -20167.073} C_VEL
LIN {X 0,Y 228.153,Z 294.69,A -85,B 0,C 180,E1 -20170.652,E2 -20170.652} C_VEL
LIN {X 0,Y 228.055,Z 294.702,A -85,B 0,C 180,E1 -20174.274,E2 -20174.274} C_VEL
LIN {X 0,Y 227.994,Z 294.71,A -85,B 0,C 180,E1 -20177.955,E2 -20177.955} C_VEL
LIN {X 0,Y 227.908,Z 294.722,A -85,B 0,C 180,E1 -20182.323,E2 -20182.323} C_VEL
LIN {X 0,Y 227.935,Z 294.72,A -85,B 0,C 180,E1 -20186.605,E2 -20186.605} C_VEL
LIN {X 0,Y 227.901,Z 294.722,A -85,B 0,C 180,E1 -20190.298,E2 -20190.298} C_VEL
LIN {X 0,Y 227.87,Z 294.724,A -85,B 0,C 180,E1 -20193.723,E2 -20193.723} C_VEL
LIN {X 0,Y 227.837,Z 294.728,A -85,B 0,C 180,E1 -20198.094,E2 -20198.094} C_VEL
LIN {X 0,Y 227.807,Z 294.731,A -85,B 0,C 180,E1 -20202.745,E2 -20202.745} C_VEL
LIN {X 0,Y 227.888,Z 294.888,A -85,B 0,C 180,E1 -20203.711,E2 -20203.711} C_VEL
LIN {X 0,Y 230.803,Z 306.7,A -85,B 0,C 180,E1 -20207.657,E2 -20207.657} C_VEL
LIN {X 0,Y 231.483,Z 308.699,A -85,B 0,C 180,E1 -20207.849,E2 -20207.849} C_VEL
LIN {X 0,Y 232.114,Z 312.47,A -85,B 0,C 180,E1 -20208.136,E2 -20208.136} C_VEL
LIN {X 0,Y 231.267,Z 325.668,A -85,B 0,C 180,E1 -20208.794,E2 -20208.794} C_VEL
LIN {X 0,Y 231.995,Z 329.4,A -85,B 0,C 180,E1 -20209.083,E2 -20209.083} C_VEL
LIN {X 0,Y 241.276,Z 355.391,A -85,B 0,C 180,E1 -20211.438,E2 -20211.438} C_VEL
LIN {X 0,Y 243.139,Z 372.64,A -85,B 0,C 180,E1 -20212.524,E2 -20212.524} C_VEL
LIN {X 0,Y 235.311,Z 474.772,A -85,B 0,C 180,E1 -20217.427,E2 -20217.427} C_VEL
LIN {X 0,Y 233.512,Z 491.51,A -85,B 0,C 180,E1 -20218.6,E2 -20218.6} C_VEL
LIN {X 0,Y 231.353,Z 508.287,A -85,B 0,C 180,E1 -20220.173,E2 -20220.173} C_VEL
LIN {X 0,Y 229.352,Z 522.687,A -85,B 0,C 180,E1 -20221.895,E2 -20221.895} C_VEL
LIN {X 0,Y 227.162,Z 536.714,A -85,B 0,C 180,E1 -20223.959,E2 -20223.959} C_VEL
LIN {X 0,Y 225.081,Z 549.758,A -85,B 0,C 180,E1 -20226.299,E2 -20226.299} C_VEL
LIN {X 0,Y 223.279,Z 561.233,A -85,B 0,C 180,E1 -20228.781,E2 -20228.781} C_VEL
LIN {X 0,Y 221.781,Z 571.876,A -85,B 0,C 180,E1 -20231.528,E2 -20231.528} C_VEL
LIN {X 0,Y 220.608,Z 582.296,A -85,B 0,C 180,E1 -20234.765,E2 -20234.765} C_VEL
LIN {X 0,Y 219.788,Z 590.827,A -85,B 0,C 180,E1 -20238.007,E2 -20238.007} C_VEL
LIN {X 0,Y 219.476,Z 596.844,A -85,B 0,C 180,E1 -20240.789,E2 -20240.789} C_VEL
LIN {X 0,Y 219.469,Z 602.343,A -85,B 0,C 180,E1 -20243.862,E2 -20243.862} C_VEL
LIN {X 0,Y 219.41,Z 607.035,A -85,B 0,C 180,E1 -20247.249,E2 -20247.249} C_VEL
LIN {X 0,Y 219.544,Z 609.874,A -85,B 0,C 180,E1 -20250.003,E2 -20250.003} C_VEL
LIN {X 0,Y 219.239,Z 611.259,A -85,B 0,C 180,E1 -20251.839,E2 -20251.839} C_VEL
LIN {X 0,Y 218.89,Z 613.081,A -85,B 0,C 180,E1 -20255.53,E2 -20255.53} C_VEL
LIN {X 0,Y 218.827,Z 613.7,A -85,B 0,C 180,E1 -20259.243,E2 -20259.243} C_VEL
LIN {X 0,Y 219.486,Z 613.154,A -85,B 0,C 180,E1 -20262.955,E2 -20262.955} C_VEL
LIN {X 0,Y 221.139,Z 611.59,A -85,B 0,C 180,E1 -20266.623,E2 -20266.623} C_VEL
LIN {X 0,Y 223.653,Z 609.006,A -85,B 0,C 180,E1 -20270.224,E2 -20270.224} C_VEL
LIN {X 0,Y 228.201,Z 604.312,A -85,B 0,C 180,E1 -20274.57,E2 -20274.57} C_VEL
LIN {X 0,Y 233.995,Z 598.013,A -85,B 0,C 180,E1 -20278.724,E2 -20278.724} C_VEL
LIN {X 0,Y 241.643,Z 589.948,A -85,B 0,C 180,E1 -20282.553,E2 -20282.553} C_VEL
LIN {X 0,Y 249.628,Z 581.192,A -85,B 0,C 180,E1 -20285.748,E2 -20285.748} C_VEL
LIN {X 0,Y 257.644,Z 572.1,A -85,B 0,C 180,E1 -20288.36,E2 -20288.36} C_VEL
LIN {X 0,Y 266.499,Z 561.585,A -85,B 0,C 180,E1 -20290.747,E2 -20290.747} C_VEL
LIN {X 0,Y 274.939,Z 550.998,A -85,B 0,C 180,E1 -20292.642,E2 -20292.642} C_VEL
LIN {X 0,Y 284.032,Z 538.905,A -85,B 0,C 180,E1 -20294.35,E2 -20294.35} C_VEL
LIN {X 0,Y 292.661,Z 526.48,A -85,B 0,C 180,E1 -20295.734,E2 -20295.734} C_VEL
LIN {X 0,Y 293.672,Z 524.992,A -85,B 0,C 180,E1 -20295.887,E2 -20295.887} C_VEL
LIN {X 0,Y 293.883,Z 524.636,A -85,B 0,C 180,E1 -20296.09,E2 -20296.09} C_VEL
LIN {X 0,Y 285.037,Z 536.658,A -85,B 0,C 180,E1 -20297.786,E2 -20297.786} C_VEL
LIN {X 0,Y 276.626,Z 547.127,A -85,B 0,C 180,E1 -20299.619,E2 -20299.619} C_VEL
LIN {X 0,Y 267.659,Z 557.397,A -85,B 0,C 180,E1 -20301.898,E2 -20301.898} C_VEL
LIN {X 0,Y 259.266,Z 566.22,A -85,B 0,C 180,E1 -20304.351,E2 -20304.351} C_VEL
LIN {X 0,Y 251.695,Z 573.61,A -85,B 0,C 180,E1 -20307.009,E2 -20307.009} C_VEL
LIN {X 0,Y 244.944,Z 579.763,A -85,B 0,C 180,E1 -20309.859,E2 -20309.859} C_VEL
LIN {X 0,Y 237.526,Z 585.806,A -85,B 0,C 180,E1 -20313.651,E2 -20313.651} C_VEL
LIN {X 0,Y 232.341,Z 589.489,A -85,B 0,C 180,E1 -20316.843,E2 -20316.843} C_VEL
LIN {X 0,Y 228.227,Z 591.989,A -85,B 0,C 180,E1 -20320.199,E2 -20320.199} C_VEL
LIN {X 0,Y 224.865,Z 593.478,A -85,B 0,C 180,E1 -20323.662,E2 -20323.662} C_VEL
LIN {X 0,Y 222.441,Z 593.936,A -85,B 0,C 180,E1 -20327.221,E2 -20327.221} C_VEL
LIN {X 0,Y 220.548,Z 593.337,A -85,B 0,C 180,E1 -20330.831,E2 -20330.831} C_VEL
LIN {X 0,Y 219.465,Z 591.582,A -85,B 0,C 180,E1 -20334.486,E2 -20334.486} C_VEL
LIN {X 0,Y 219.03,Z 588.696,A -85,B 0,C 180,E1 -20338.16,E2 -20338.16} C_VEL
LIN {X 0,Y 218.832,Z 584.575,A -85,B 0,C 180,E1 -20341.839,E2 -20341.839} C_VEL
LIN {X 0,Y 218.932,Z 579.081,A -85,B 0,C 180,E1 -20345.525,E2 -20345.525} C_VEL
LIN {X 0,Y 219.363,Z 572.033,A -85,B 0,C 180,E1 -20349.216,E2 -20349.216} C_VEL
LIN {X 0,Y 220.036,Z 564.42,A -85,B 0,C 180,E1 -20352.449,E2 -20352.449} C_VEL
LIN {X 0,Y 221.234,Z 555.258,A -85,B 0,C 180,E1 -20355.664,E2 -20355.664} C_VEL
LIN {X 0,Y 222.691,Z 544.595,A -85,B 0,C 180,E1 -20358.771,E2 -20358.771} C_VEL
LIN {X 0,Y 224.439,Z 532.961,A -85,B 0,C 180,E1 -20361.587,E2 -20361.587} C_VEL
LIN {X 0,Y 226.324,Z 520.784,A -85,B 0,C 180,E1 -20364.05,E2 -20364.05} C_VEL
LIN {X 0,Y 228.447,Z 506.647,A -85,B 0,C 180,E1 -20366.427,E2 -20366.427} C_VEL
LIN {X 0,Y 230.565,Z 491.991,A -85,B 0,C 180,E1 -20368.441,E2 -20368.441} C_VEL
LIN {X 0,Y 232.534,Z 476.433,A -85,B 0,C 180,E1 -20370.161,E2 -20370.161} C_VEL
LIN {X 0,Y 234.266,Z 459.597,A -85,B 0,C 180,E1 -20371.603,E2 -20371.603} C_VEL
LIN {X 0,Y 235.815,Z 442.215,A -85,B 0,C 180,E1 -20372.694,E2 -20372.694} C_VEL
LIN {X 0,Y 242.919,Z 347.235,A -85,B 0,C 180,E1 -20377.174,E2 -20377.174} C_VEL
LIN {X 0,Y 227.43,Z 311.058,A -85,B 0,C 180,E1 -20380.754,E2 -20380.754} C_VEL
LIN {X 0,Y 220.89,Z 296.316,A -85,B 0,C 180,E1 -20382.386,E2 -20382.386} C_VEL
LIN {X 0,Y 220.787,Z 295.61,A -85,B 0,C 180,E1 -20382.515,E2 -20382.515} C_VEL
LIN {X 0,Y 220.766,Z 295.61,A -85,B 0,C 180,E1 -20387.068,E2 -20387.068} C_VEL
LIN {X 0,Y 220.806,Z 295.603,A -85,B 0,C 180,E1 -20390.46,E2 -20390.46} C_VEL
LIN {X 0,Y 220.8,Z 295.604,A -85,B 0,C 180,E1 -20395.042,E2 -20395.042} C_VEL
LIN {X 0,Y 220.832,Z 295.6,A -85,B 0,C 180,E1 -20399.387,E2 -20399.387} C_VEL
LIN {X 0,Y 220.873,Z 295.598,A -85,B 0,C 180,E1 -20403.544,E2 -20403.544} C_VEL
LIN {X 0,Y 220.863,Z 295.599,A -85,B 0,C 180,E1 -20407.549,E2 -20407.549} C_VEL
LIN {X 0,Y 220.924,Z 295.59,A -85,B 0,C 180,E1 -20412.615,E2 -20412.615} C_VEL
LIN {X 0,Y 220.999,Z 295.581,A -85,B 0,C 180,E1 -20417.135,E2 -20417.135} C_VEL
LIN {X 0,Y 221.231,Z 295.553,A -85,B 0,C 180,E1 -20420.858,E2 -20420.858} C_VEL
LIN {X 0,Y 221.284,Z 295.545,A -85,B 0,C 180,E1 -20422.699,E2 -20422.699} C_VEL
LIN {X 0,Y 221.505,Z 295.517,A -85,B 0,C 180,E1 -20428.179,E2 -20428.179} C_VEL
LIN {X 0,Y 221.505,Z 295.516,A -85,B 0,C 180,E1 -20431.816,E2 -20431.816} C_VEL
LIN {X 0,Y 221.298,Z 295.545,A -85,B 0,C 180,E1 -20437.296,E2 -20437.296} C_VEL
LIN {X 0,Y 221.098,Z 295.565,A -85,B 0,C 180,E1 -20440.992,E2 -20440.992} C_VEL
LIN {X 0,Y 221.007,Z 295.578,A -85,B 0,C 180,E1 -20446.628,E2 -20446.628} C_VEL
LIN {X 0,Y 220.883,Z 295.593,A -85,B 0,C 180,E1 -20450.484,E2 -20450.484} C_VEL
LIN {X 0,Y 220.857,Z 295.597,A -85,B 0,C 180,E1 -20454.433,E2 -20454.433} C_VEL
LIN {X 0,Y 220.816,Z 295.601,A -85,B 0,C 180,E1 -20458.513,E2 -20458.513} C_VEL
LIN {X 0,Y 220.811,Z 295.603,A -85,B 0,C 180,E1 -20462.754,E2 -20462.754} C_VEL
LIN {X 0,Y 220.827,Z 295.602,A -85,B 0,C 180,E1 -20467.287,E2 -20467.287} C_VEL
LIN {X 0,Y 220.758,Z 295.609,A -85,B 0,C 180,E1 -20471.951,E2 -20471.951} C_VEL
LIN {X 0,Y 220.763,Z 295.61,A -85,B 0,C 180,E1 -20475.546,E2 -20475.546} C_VEL
LIN {X 0,Y 220.794,Z 295.604,A -85,B 0,C 180,E1 -20480.463,E2 -20480.463} C_VEL
LIN {X 0,Y 220.788,Z 295.607,A -85,B 0,C 180,E1 -20485.045,E2 -20485.045} C_VEL
LIN {X 0,Y 220.855,Z 295.597,A -85,B 0,C 180,E1 -20489.395,E2 -20489.395} C_VEL
LIN {X 0,Y 220.882,Z 295.595,A -85,B 0,C 180,E1 -20493.55,E2 -20493.55} C_VEL
LIN {X 0,Y 220.853,Z 295.597,A -85,B 0,C 180,E1 -20497.552,E2 -20497.552} C_VEL
LIN {X 0,Y 220.972,Z 295.583,A -85,B 0,C 180,E1 -20502.572,E2 -20502.572} C_VEL
LIN {X 0,Y 221.014,Z 295.578,A -85,B 0,C 180,E1 -20507.14,E2 -20507.14} C_VEL
LIN {X 0,Y 221.224,Z 295.553,A -85,B 0,C 180,E1 -20510.862,E2 -20510.862} C_VEL
LIN {X 0,Y 221.276,Z 295.547,A -85,B 0,C 180,E1 -20512.703,E2 -20512.703} C_VEL
LIN {X 0,Y 221.501,Z 295.516,A -85,B 0,C 180,E1 -20518.183,E2 -20518.183} C_VEL
LIN {X 0,Y 221.501,Z 295.516,A -85,B 0,C 180,E1 -20521.82,E2 -20521.82} C_VEL
LIN {X 0,Y 221.279,Z 295.546,A -85,B 0,C 180,E1 -20527.3,E2 -20527.3} C_VEL
LIN {X 0,Y 221.102,Z 295.57,A -85,B 0,C 180,E1 -20530.996,E2 -20530.996} C_VEL
LIN {X 0,Y 221.007,Z 295.581,A -85,B 0,C 180,E1 -20536.632,E2 -20536.632} C_VEL
LIN {X 0,Y 220.875,Z 295.599,A -85,B 0,C 180,E1 -20540.489,E2 -20540.489} C_VEL
LIN {X 0,Y 220.854,Z 295.601,A -85,B 0,C 180,E1 -20544.438,E2 -20544.438} C_VEL
LIN {X 0,Y 220.829,Z 295.605,A -85,B 0,C 180,E1 -20548.516,E2 -20548.516} C_VEL
LIN {X 0,Y 220.811,Z 295.607,A -85,B 0,C 180,E1 -20552.758,E2 -20552.758} C_VEL
LIN {X 0,Y 220.804,Z 295.605,A -85,B 0,C 180,E1 -20557.281,E2 -20557.281} C_VEL
LIN {X 0,Y 220.765,Z 295.607,A -85,B 0,C 180,E1 -20561.955,E2 -20561.955} C_VEL
LIN {X 0,Y 220.815,Z 295.723,A -85,B 0,C 180,E1 -20563.124,E2 -20563.124} C_VEL
LIN {X 0,Y 223.394,Z 306.266,A -85,B 0,C 180,E1 -20566.762,E2 -20566.762} C_VEL
LIN {X 0,Y 231.995,Z 329.4,A -85,B 0,C 180,E1 -20569.083,E2 -20569.083} C_VEL
LIN {X 0,Y 233.452,Z 334.808,A -85,B 0,C 180,E1 -20569.537,E2 -20569.537} C_VEL
LIN {X 0,Y 234.302,Z 344.316,A -85,B 0,C 180,E1 -20570.155,E2 -20570.155} C_VEL
LIN {X 0,Y 234.436,Z 352.106,A -85,B 0,C 180,E1 -20570.604,E2 -20570.604} C_VEL
LIN {X 0,Y 234.974,Z 359.83,A -85,B 0,C 180,E1 -20571.087,E2 -20571.087} C_VEL
LIN {X 0,Y 236.377,Z 373.799,A -85,B 0,C 180,E1 -20571.988,E2 -20571.988} C_VEL
LIN {X 0,Y 228.461,Z 473.89,A -85,B 0,C 180,E1 -20576.974,E2 -20576.974} C_VEL
LIN {X 0,Y 226.629,Z 490.769,A -85,B 0,C 180,E1 -20578.188,E2 -20578.188} C_VEL
LIN {X 0,Y 224.439,Z 507.523,A -85,B 0,C 180,E1 -20579.806,E2 -20579.806} C_VEL
LIN {X 0,Y 222.279,Z 522.754,A -85,B 0,C 180,E1 -20581.691,E2 -20581.691} C_VEL
LIN {X 0,Y 219.992,Z 537.392,A -85,B 0,C 180,E1 -20583.946,E2 -20583.946} C_VEL
LIN {X 0,Y 217.769,Z 550.683,A -85,B 0,C 180,E1 -20586.464,E2 -20586.464} C_VEL
LIN {X 0,Y 216.016,Z 561.979,A -85,B 0,C 180,E1 -20589.033,E2 -20589.033} C_VEL
LIN {X 0,Y 214.535,Z 572.214,A -85,B 0,C 180,E1 -20591.811,E2 -20591.811} C_VEL
LIN {X 0,Y 213.576,Z 581.291,A -85,B 0,C 180,E1 -20594.74,E2 -20594.74} C_VEL
LIN {X 0,Y 212.772,Z 589.904,A -85,B 0,C 180,E1 -20598.089,E2 -20598.089} C_VEL
LIN {X 0,Y 212.469,Z 596.916,A -85,B 0,C 180,E1 -20601.442,E2 -20601.442} C_VEL
LIN {X 0,Y 212.464,Z 601.791,A -85,B 0,C 180,E1 -20604.308,E2 -20604.308} C_VEL
LIN {X 0,Y 212.459,Z 606.794,A -85,B 0,C 180,E1 -20608.107,E2 -20608.107} C_VEL
LIN {X 0,Y 212.524,Z 608.716,A -85,B 0,C 180,E1 -20610.003,E2 -20610.003} C_VEL
LIN {X 0,Y 212.229,Z 610.227,A -85,B 0,C 180,E1 -20611.9,E2 -20611.9} C_VEL
LIN {X 0,Y 211.826,Z 612.241,A -85,B 0,C 180,E1 -20615.715,E2 -20615.715} C_VEL
LIN {X 0,Y 211.8,Z 613.025,A -85,B 0,C 180,E1 -20619.553,E2 -20619.553} C_VEL
LIN {X 0,Y 212.523,Z 612.758,A -85,B 0,C 180,E1 -20623.387,E2 -20623.387} C_VEL
LIN {X 0,Y 214.278,Z 611.445,A -85,B 0,C 180,E1 -20627.171,E2 -20627.171} C_VEL
LIN {X 0,Y 216.96,Z 609.093,A -85,B 0,C 180,E1 -20630.877,E2 -20630.877} C_VEL
LIN {X 0,Y 221.756,Z 604.781,A -85,B 0,C 180,E1 -20635.334,E2 -20635.334} C_VEL
LIN {X 0,Y 227.86,Z 598.934,A -85,B 0,C 180,E1 -20639.573,E2 -20639.573} C_VEL
LIN {X 0,Y 235.624,Z 591.625,A -85,B 0,C 180,E1 -20643.366,E2 -20643.366} C_VEL
LIN {X 0,Y 243.15,Z 584.206,A -85,B 0,C 180,E1 -20646.339,E2 -20646.339} C_VEL
LIN {X 0,Y 252.389,Z 574.701,A -85,B 0,C 180,E1 -20649.311,E2 -20649.311} C_VEL
LIN {X 0,Y 261.533,Z 564.858,A -85,B 0,C 180,E1 -20651.692,E2 -20651.692} C_VEL
LIN {X 0,Y 270.184,Z 555.054,A -85,B 0,C 180,E1 -20653.578,E2 -20653.578} C_VEL
LIN {X 0,Y 280.348,Z 542.751,A -85,B 0,C 180,E1 -20655.417,E2 -20655.417} C_VEL
LIN {X 0,Y 283.617,Z 538.535,A -85,B 0,C 180,E1 -20655.943,E2 -20655.943} C_VEL
LIN {X 0,Y 284.49,Z 537.383,A -85,B 0,C 180,E1 -20656.234,E2 -20656.234} C_VEL
LIN {X 0,Y 276.105,Z 547.179,A -85,B 0,C 180,E1 -20657.879,E2 -20657.879} C_VEL
LIN {X 0,Y 266.133,Z 557.831,A -85,B 0,C 180,E1 -20660.178,E2 -20660.178} C_VEL
LIN {X 0,Y 258.299,Z 565.557,A -85,B 0,C 180,E1 -20662.25,E2 -20662.25} C_VEL
LIN {X 0,Y 250.461,Z 572.671,A -85,B 0,C 180,E1 -20664.661,E2 -20664.661} C_VEL
LIN {X 0,Y 242.576,Z 579.319,A -85,B 0,C 180,E1 -20667.588,E2 -20667.588} C_VEL
LIN {X 0,Y 235.908,Z 584.451,A -85,B 0,C 180,E1 -20670.556,E2 -20670.556} C_VEL
LIN {X 0,Y 228.488,Z 589.405,A -85,B 0,C 180,E1 -20674.492,E2 -20674.492} C_VEL
LIN {X 0,Y 223.713,Z 592.135,A -85,B 0,C 180,E1 -20677.852,E2 -20677.852} C_VEL
LIN {X 0,Y 219.711,Z 593.887,A -85,B 0,C 180,E1 -20681.343,E2 -20681.343} C_VEL
LIN {X 0,Y 216.724,Z 594.537,A -85,B 0,C 180,E1 -20684.963,E2 -20684.963} C_VEL
LIN {X 0,Y 214.456,Z 594.174,A -85,B 0,C 180,E1 -20688.659,E2 -20688.659} C_VEL
LIN {X 0,Y 212.89,Z 592.763,A -85,B 0,C 180,E1 -20692.411,E2 -20692.411} C_VEL
LIN {X 0,Y 212.151,Z 590.242,A -85,B 0,C 180,E1 -20696.2,E2 -20696.2} C_VEL
LIN {X 0,Y 211.817,Z 586.489,A -85,B 0,C 180,E1 -20699.999,E2 -20699.999} C_VEL
LIN {X 0,Y 211.758,Z 581.431,A -85,B 0,C 180,E1 -20703.804,E2 -20703.804} C_VEL
LIN {X 0,Y 212.06,Z 574.877,A -85,B 0,C 180,E1 -20707.632,E2 -20707.632} C_VEL
LIN {X 0,Y 212.594,Z 567.805,A -85,B 0,C 180,E1 -20710.956,E2 -20710.956} C_VEL
LIN {X 0,Y 213.588,Z 559.248,A -85,B 0,C 180,E1 -20714.286,E2 -20714.286} C_VEL
LIN {X 0,Y 214.929,Z 548.965,A -85,B 0,C 180,E1 -20717.603,E2 -20717.603} C_VEL
LIN {X 0,Y 216.494,Z 538.479,A -85,B 0,C 180,E1 -20720.422,E2 -20720.422} C_VEL
LIN {X 0,Y 218.475,Z 526.127,A -85,B 0,C 180,E1 -20723.206,E2 -20723.206} C_VEL
LIN {X 0,Y 220.494,Z 512.619,A -85,B 0,C 180,E1 -20725.738,E2 -20725.738} C_VEL
LIN {X 0,Y 222.689,Z 498.514,A -85,B 0,C 180,E1 -20727.908,E2 -20727.908} C_VEL
LIN {X 0,Y 224.666,Z 483.628,A -85,B 0,C 180,E1 -20729.773,E2 -20729.773} C_VEL
LIN {X 0,Y 226.508,Z 468.207,A -85,B 0,C 180,E1 -20731.311,E2 -20731.311} C_VEL
LIN {X 0,Y 228.164,Z 451.131,A -85,B 0,C 180,E1 -20732.617,E2 -20732.617} C_VEL
LIN {X 0,Y 229.889,Z 428.495,A -85,B 0,C 180,E1 -20733.853,E2 -20733.853} C_VEL
LIN {X 0,Y 236.201,Z 348.958,A -85,B 0,C 180,E1 -20737.708,E2 -20737.708} C_VEL
LIN {X 0,Y 220.833,Z 312.991,A -85,B 0,C 180,E1 -20741.389,E2 -20741.389} C_VEL
LIN {X 0,Y 213.875,Z 297.334,A -85,B 0,C 180,E1 -20743.187,E2 -20743.187} C_VEL
LIN {X 0,Y 213.728,Z 296.488,A -85,B 0,C 180,E1 -20743.317,E2 -20743.317} C_VEL
LIN {X 0,Y 213.706,Z 296.491,A -85,B 0,C 180,E1 -20746.341,E2 -20746.341} C_VEL
LIN {X 0,Y 213.717,Z 296.488,A -85,B 0,C 180,E1 -20749.14,E2 -20749.14} C_VEL
LIN {X 0,Y 213.743,Z 296.486,A -85,B 0,C 180,E1 -20753.709,E2 -20753.709} C_VEL
LIN {X 0,Y 213.757,Z 296.481,A -85,B 0,C 180,E1 -20758.258,E2 -20758.258} C_VEL
LIN {X 0,Y 213.786,Z 296.478,A -85,B 0,C 180,E1 -20762.595,E2 -20762.595} C_VEL
LIN {X 0,Y 213.807,Z 296.476,A -85,B 0,C 180,E1 -20766.977,E2 -20766.977} C_VEL
LIN {X 0,Y 213.887,Z 296.467,A -85,B 0,C 180,E1 -20772.796,E2 -20772.796} C_VEL
LIN {X 0,Y 213.937,Z 296.46,A -85,B 0,C 180,E1 -20776.703,E2 -20776.703} C_VEL
LIN {X 0,Y 214.163,Z 296.433,A -85,B 0,C 180,E1 -20780.554,E2 -20780.554} C_VEL
LIN {X 0,Y 214.222,Z 296.424,A -85,B 0,C 180,E1 -20782.457,E2 -20782.457} C_VEL
LIN {X 0,Y 214.438,Z 296.398,A -85,B 0,C 180,E1 -20788.119,E2 -20788.119} C_VEL
LIN {X 0,Y 214.544,Z 296.383,A -85,B 0,C 180,E1 -20789.997,E2 -20789.997} C_VEL
LIN {X 0,Y 214.438,Z 296.396,A -85,B 0,C 180,E1 -20791.876,E2 -20791.876} C_VEL
LIN {X 0,Y 214.233,Z 296.425,A -85,B 0,C 180,E1 -20797.538,E2 -20797.538} C_VEL
LIN {X 0,Y 214.015,Z 296.449,A -85,B 0,C 180,E1 -20801.361,E2 -20801.361} C_VEL
LIN {X 0,Y 213.925,Z 296.463,A -85,B 0,C 180,E1 -20805.235,E2 -20805.235} C_VEL
LIN {X 0,Y 213.83,Z 296.471,A -85,B 0,C 180,E1 -20809.185,E2 -20809.185} C_VEL
LIN {X 0,Y 213.837,Z 296.474,A -85,B 0,C 180,E1 -20813.225,E2 -20813.225} C_VEL
LIN {X 0,Y 213.818,Z 296.474,A -85,B 0,C 180,E1 -20817.448,E2 -20817.448} C_VEL
LIN {X 0,Y 213.759,Z 296.483,A -85,B 0,C 180,E1 -20821.736,E2 -20821.736} C_VEL
LIN {X 0,Y 213.737,Z 296.482,A -85,B 0,C 180,E1 -20826.286,E2 -20826.286} C_VEL
LIN {X 0,Y 213.7,Z 296.491,A -85,B 0,C 180,E1 -20831.124,E2 -20831.124} C_VEL
LIN {X 0,Y 213.695,Z 296.488,A -85,B 0,C 180,E1 -20833.677,E2 -20833.677} C_VEL
LIN {X 0,Y 213.695,Z 296.489,A -85,B 0,C 180,E1 -20836.343,E2 -20836.343} C_VEL
LIN {X 0,Y 213.705,Z 296.491,A -85,B 0,C 180,E1 -20839.142,E2 -20839.142} C_VEL
LIN {X 0,Y 213.731,Z 296.485,A -85,B 0,C 180,E1 -20843.711,E2 -20843.711} C_VEL
LIN {X 0,Y 213.782,Z 296.479,A -85,B 0,C 180,E1 -20848.725,E2 -20848.725} C_VEL
LIN {X 0,Y 213.814,Z 296.474,A -85,B 0,C 180,E1 -20852.603,E2 -20852.603} C_VEL
LIN {X 0,Y 213.807,Z 296.478,A -85,B 0,C 180,E1 -20856.974,E2 -20856.974} C_VEL
LIN {X 0,Y 213.931,Z 296.461,A -85,B 0,C 180,E1 -20862.804,E2 -20862.804} C_VEL
LIN {X 0,Y 213.968,Z 296.455,A -85,B 0,C 180,E1 -20866.709,E2 -20866.709} C_VEL
LIN {X 0,Y 214.155,Z 296.432,A -85,B 0,C 180,E1 -20870.557,E2 -20870.557} C_VEL
LIN {X 0,Y 214.215,Z 296.425,A -85,B 0,C 180,E1 -20872.461,E2 -20872.461} C_VEL
LIN {X 0,Y 214.434,Z 296.397,A -85,B 0,C 180,E1 -20878.123,E2 -20878.123} C_VEL
LIN {X 0,Y 214.539,Z 296.384,A -85,B 0,C 180,E1 -20880.001,E2 -20880.001} C_VEL
LIN {X 0,Y 214.434,Z 296.397,A -85,B 0,C 180,E1 -20881.88,E2 -20881.88} C_VEL
LIN {X 0,Y 214.217,Z 296.425,A -85,B 0,C 180,E1 -20887.542,E2 -20887.542} C_VEL
LIN {X 0,Y 214.035,Z 296.449,A -85,B 0,C 180,E1 -20891.364,E2 -20891.364} C_VEL
LIN {X 0,Y 213.924,Z 296.464,A -85,B 0,C 180,E1 -20895.239,E2 -20895.239} C_VEL
LIN {X 0,Y 213.827,Z 296.477,A -85,B 0,C 180,E1 -20899.19,E2 -20899.19} C_VEL
LIN {X 0,Y 213.803,Z 296.48,A -85,B 0,C 180,E1 -20903.233,E2 -20903.233} C_VEL
LIN {X 0,Y 213.822,Z 296.477,A -85,B 0,C 180,E1 -20907.452,E2 -20907.452} C_VEL
LIN {X 0,Y 213.77,Z 296.481,A -85,B 0,C 180,E1 -20911.739,E2 -20911.739} C_VEL
LIN {X 0,Y 213.737,Z 296.485,A -85,B 0,C 180,E1 -20916.291,E2 -20916.291} C_VEL
LIN {X 0,Y 213.707,Z 296.487,A -85,B 0,C 180,E1 -20921.128,E2 -20921.128} C_VEL
LIN {X 0,Y 213.747,Z 296.628,A -85,B 0,C 180,E1 -20922.541,E2 -20922.541} C_VEL
LIN {X 0,Y 216.044,Z 305.859,A -85,B 0,C 180,E1 -20925.847,E2 -20925.847} C_VEL
LIN {X 0,Y 229.452,Z 342.299,A -85,B 0,C 180,E1 -20929.55,E2 -20929.55} C_VEL
LIN {X 0,Y 234.796,Z 357.67,A -85,B 0,C 180,E1 -20930.95,E2 -20930.95} C_VEL
LIN {X 0,Y 234.974,Z 359.83,A -85,B 0,C 180,E1 -20931.087,E2 -20931.087} C_VEL
LIN {X 0,Y 235.097,Z 363.646,A -85,B 0,C 180,E1 -20931.31,E2 -20931.31} C_VEL
LIN {X 0,Y 234.605,Z 367.494,A -85,B 0,C 180,E1 -20931.478,E2 -20931.478} C_VEL
LIN {X 0,Y 232.501,Z 375.112,A -85,B 0,C 180,E1 -20931.713,E2 -20931.713} C_VEL
LIN {X 0,Y 228.945,Z 386.647,A -85,B 0,C 180,E1 -20932.049,E2 -20932.049} C_VEL
LIN {X 0,Y 228.326,Z 390.572,A -85,B 0,C 180,E1 -20932.218,E2 -20932.218} C_VEL
LIN {X 0,Y 221.569,Z 473.673,A -85,B 0,C 180,E1 -20936.559,E2 -20936.559} C_VEL
LIN {X 0,Y 219.651,Z 491.023,A -85,B 0,C 180,E1 -20937.867,E2 -20937.867} C_VEL
LIN {X 0,Y 217.414,Z 507.593,A -85,B 0,C 180,E1 -20939.532,E2 -20939.532} C_VEL
LIN {X 0,Y 215.206,Z 522.693,A -85,B 0,C 180,E1 -20941.475,E2 -20941.475} C_VEL
LIN {X 0,Y 212.886,Z 537.191,A -85,B 0,C 180,E1 -20943.8,E2 -20943.8} C_VEL
LIN {X 0,Y 210.674,Z 550.418,A -85,B 0,C 180,E1 -20946.405,E2 -20946.405} C_VEL
LIN {X 0,Y 208.797,Z 562.584,A -85,B 0,C 180,E1 -20949.306,E2 -20949.306} C_VEL
LIN {X 0,Y 207.306,Z 572.829,A -85,B 0,C 180,E1 -20952.238,E2 -20952.238} C_VEL
LIN {X 0,Y 206.419,Z 581.576,A -85,B 0,C 180,E1 -20955.208,E2 -20955.208} C_VEL
LIN {X 0,Y 205.711,Z 590.032,A -85,B 0,C 180,E1 -20958.674,E2 -20958.674} C_VEL
LIN {X 0,Y 205.471,Z 596.923,A -85,B 0,C 180,E1 -20962.139,E2 -20962.139} C_VEL
LIN {X 0,Y 205.447,Z 601.637,A -85,B 0,C 180,E1 -20965.097,E2 -20965.097} C_VEL
LIN {X 0,Y 205.475,Z 606.494,A -85,B 0,C 180,E1 -20969.023,E2 -20969.023} C_VEL
LIN {X 0,Y 205.514,Z 607.486,A -85,B 0,C 180,E1 -20970.003,E2 -20970.003} C_VEL
LIN {X 0,Y 205.215,Z 609.08,A -85,B 0,C 180,E1 -20971.965,E2 -20971.965} C_VEL
LIN {X 0,Y 204.797,Z 611.292,A -85,B 0,C 180,E1 -20975.912,E2 -20975.912} C_VEL
LIN {X 0,Y 204.758,Z 612.34,A -85,B 0,C 180,E1 -20979.884,E2 -20979.884} C_VEL
LIN {X 0,Y 205.576,Z 612.289,A -85,B 0,C 180,E1 -20983.848,E2 -20983.848} C_VEL
LIN {X 0,Y 208.31,Z 610.621,A -85,B 0,C 180,E1 -20989.146,E2 -20989.146} C_VEL
LIN {X 0,Y 212.144,Z 607.789,A -85,B 0,C 180,E1 -20993.427,E2 -20993.427} C_VEL
LIN {X 0,Y 217.749,Z 603.273,A -85,B 0,C 180,E1 -20997.907,E2 -20997.907} C_VEL
LIN {X 0,Y 223.314,Z 598.578,A -85,B 0,C 180,E1 -21001.286,E2 -21001.286} C_VEL
LIN {X 0,Y 231.891,Z 591.273,A -85,B 0,C 180,E1 -21005.161,E2 -21005.161} C_VEL
LIN {X 0,Y 241.769,Z 582.359,A -85,B 0,C 180,E1 -21008.683,E2 -21008.683} C_VEL
LIN {X 0,Y 251.806,Z 572.82,A -85,B 0,C 180,E1 -21011.522,E2 -21011.522} C_VEL
LIN {X 0,Y 262.871,Z 561.665,A -85,B 0,C 180,E1 -21014.04,E2 -21014.04} C_VEL
LIN {X 0,Y 273.554,Z 550.115,A -85,B 0,C 180,E1 -21016.004,E2 -21016.004} C_VEL
LIN {X 0,Y 274.948,Z 548.545,A -85,B 0,C 180,E1 -21016.357,E2 -21016.357} C_VEL
LIN {X 0,Y 264.934,Z 558.514,A -85,B 0,C 180,E1 -21018.456,E2 -21018.456} C_VEL
LIN {X 0,Y 255.496,Z 567.111,A -85,B 0,C 180,E1 -21020.752,E2 -21020.752} C_VEL
LIN {X 0,Y 246.748,Z 574.405,A -85,B 0,C 180,E1 -21023.263,E2 -21023.263} C_VEL
LIN {X 0,Y 238.833,Z 580.45,A -85,B 0,C 180,E1 -21026.005,E2 -21026.005} C_VEL
LIN {X 0,Y 230.015,Z 586.534,A -85,B 0,C 180,E1 -21029.724,E2 -21029.724} C_VEL
LIN {X 0,Y 222.266,Z 591.009,A -85,B 0,C 180,E1 -21033.724,E2 -21033.724} C_VEL
LIN {X 0,Y 217.257,Z 593.384,A -85,B 0,C 180,E1 -21037.157,E2 -21037.157} C_VEL
LIN {X 0,Y 213.043,Z 594.779,A -85,B 0,C 180,E1 -21040.737,E2 -21040.737} C_VEL
LIN {X 0,Y 209.91,Z 595.184,A -85,B 0,C 180,E1 -21044.462,E2 -21044.462} C_VEL
LIN {X 0,Y 207.508,Z 594.557,A -85,B 0,C 180,E1 -21048.274,E2 -21048.274} C_VEL
LIN {X 0,Y 205.857,Z 592.848,A -85,B 0,C 180,E1 -21052.15,E2 -21052.15} C_VEL
LIN {X 0,Y 205.076,Z 590.055,A -85,B 0,C 180,E1 -21056.068,E2 -21056.068} C_VEL
LIN {X 0,Y 204.749,Z 586.081,A -85,B 0,C 180,E1 -21059.998,E2 -21059.998} C_VEL
LIN {X 0,Y 204.685,Z 580.771,A -85,B 0,C 180,E1 -21063.936,E2 -21063.936} C_VEL
LIN {X 0,Y 205.008,Z 573.96,A -85,B 0,C 180,E1 -21067.88,E2 -21067.88} C_VEL
LIN {X 0,Y 205.587,Z 566.583,A -85,B 0,C 180,E1 -21071.334,E2 -21071.334} C_VEL
LIN {X 0,Y 206.692,Z 557.721,A -85,B 0,C 180,E1 -21074.773,E2 -21074.773} C_VEL
LIN {X 0,Y 208.068,Z 547.23,A -85,B 0,C 180,E1 -21078.14,E2 -21078.14} C_VEL
LIN {X 0,Y 209.93,Z 535.131,A -85,B 0,C 180,E1 -21081.349,E2 -21081.349} C_VEL
LIN {X 0,Y 212.041,Z 522.078,A -85,B 0,C 180,E1 -21084.213,E2 -21084.213} C_VEL
LIN {X 0,Y 214.238,Z 507.674,A -85,B 0,C 180,E1 -21086.81,E2 -21086.81} C_VEL
LIN {X 0,Y 216.375,Z 493.453,A -85,B 0,C 180,E1 -21088.906,E2 -21088.906} C_VEL
LIN {X 0,Y 218.539,Z 477.287,A -85,B 0,C 180,E1 -21090.831,E2 -21090.831} C_VEL
LIN {X 0,Y 220.385,Z 460.786,A -85,B 0,C 180,E1 -21092.352,E2 -21092.352} C_VEL
LIN {X 0,Y 221.918,Z 443.777,A -85,B 0,C 180,E1 -21093.518,E2 -21093.518} C_VEL
LIN {X 0,Y 229.465,Z 350.682,A -85,B 0,C 180,E1 -21098.257,E2 -21098.257} C_VEL
LIN {X 0,Y 214.632,Z 315.789,A -85,B 0,C 180,E1 -21101.931,E2 -21101.931} C_VEL
LIN {X 0,Y 206.727,Z 297.839,A -85,B 0,C 180,E1 -21104.071,E2 -21104.071} C_VEL
LIN {X 0,Y 206.639,Z 297.373,A -85,B 0,C 180,E1 -21104.139,E2 -21104.139} C_VEL
LIN {X 0,Y 206.642,Z 297.369,A -85,B 0,C 180,E1 -21108.434,E2 -21108.434} C_VEL
LIN {X 0,Y 206.68,Z 297.366,A -85,B 0,C 180,E1 -21112.257,E2 -21112.257} C_VEL
LIN {X 0,Y 206.694,Z 297.364,A -85,B 0,C 180,E1 -21117.039,E2 -21117.039} C_VEL
LIN {X 0,Y 206.707,Z 297.361,A -85,B 0,C 180,E1 -21122.124,E2 -21122.124} C_VEL
LIN {X 0,Y 206.742,Z 297.355,A -85,B 0,C 180,E1 -21126.607,E2 -21126.607} C_VEL
LIN {X 0,Y 206.821,Z 297.348,A -85,B 0,C 180,E1 -21132.189,E2 -21132.189} C_VEL
LIN {X 0,Y 206.876,Z 297.341,A -85,B 0,C 180,E1 -21136.24,E2 -21136.24} C_VEL
LIN {X 0,Y 207.101,Z 297.314,A -85,B 0,C 180,E1 -21140.228,E2 -21140.228} C_VEL
LIN {X 0,Y 207.163,Z 297.304,A -85,B 0,C 180,E1 -21142.198,E2 -21142.198} C_VEL
LIN {X 0,Y 207.375,Z 297.278,A -85,B 0,C 180,E1 -21148.055,E2 -21148.055} C_VEL
LIN {X 0,Y 207.508,Z 297.259,A -85,B 0,C 180,E1 -21149.997,E2 -21149.997} C_VEL
LIN {X 0,Y 207.375,Z 297.275,A -85,B 0,C 180,E1 -21151.939,E2 -21151.939} C_VEL
LIN {X 0,Y 207.17,Z 297.303,A -85,B 0,C 180,E1 -21157.796,E2 -21157.796} C_VEL
LIN {X 0,Y 206.935,Z 297.333,A -85,B 0,C 180,E1 -21161.755,E2 -21161.755} C_VEL
LIN {X 0,Y 206.858,Z 297.342,A -85,B 0,C 180,E1 -21165.768,E2 -21165.768} C_VEL
LIN {X 0,Y 206.774,Z 297.351,A -85,B 0,C 180,E1 -21169.867,E2 -21169.867} C_VEL
LIN {X 0,Y 206.753,Z 297.354,A -85,B 0,C 180,E1 -21174.07,E2 -21174.07} C_VEL
LIN {X 0,Y 206.726,Z 297.356,A -85,B 0,C 180,E1 -21178.418,E2 -21178.418} C_VEL
LIN {X 0,Y 206.694,Z 297.363,A -85,B 0,C 180,E1 -21182.955,E2 -21182.955} C_VEL
LIN {X 0,Y 206.711,Z 297.359,A -85,B 0,C 180,E1 -21185.319,E2 -21185.319} C_VEL
LIN {X 0,Y 206.651,Z 297.367,A -85,B 0,C 180,E1 -21190.249,E2 -21190.249} C_VEL
LIN {X 0,Y 206.622,Z 297.372,A -85,B 0,C 180,E1 -21195.581,E2 -21195.581} C_VEL
LIN {X 0,Y 206.648,Z 297.367,A -85,B 0,C 180,E1 -21199.748,E2 -21199.748} C_VEL
LIN {X 0,Y 206.686,Z 297.362,A -85,B 0,C 180,E1 -21204.688,E2 -21204.688} C_VEL
LIN {X 0,Y 206.711,Z 297.359,A -85,B 0,C 180,E1 -21209.339,E2 -21209.339} C_VEL
LIN {X 0,Y 206.719,Z 297.359,A -85,B 0,C 180,E1 -21213.772,E2 -21213.772} C_VEL
LIN {X 0,Y 206.726,Z 297.355,A -85,B 0,C 180,E1 -21218.042,E2 -21218.042} C_VEL
LIN {X 0,Y 206.86,Z 297.34,A -85,B 0,C 180,E1 -21222.197,E2 -21222.197} C_VEL
LIN {X 0,Y 206.902,Z 297.334,A -85,B 0,C 180,E1 -21226.246,E2 -21226.246} C_VEL
LIN {X 0,Y 207.094,Z 297.311,A -85,B 0,C 180,E1 -21230.232,E2 -21230.232} C_VEL
LIN {X 0,Y 207.155,Z 297.304,A -85,B 0,C 180,E1 -21232.202,E2 -21232.202} C_VEL
LIN {X 0,Y 207.371,Z 297.277,A -85,B 0,C 180,E1 -21238.059,E2 -21238.059} C_VEL
LIN {X 0,Y 207.504,Z 297.26,A -85,B 0,C 180,E1 -21240.002,E2 -21240.002} C_VEL
LIN {X 0,Y 207.371,Z 297.277,A -85,B 0,C 180,E1 -21241.944,E2 -21241.944} C_VEL
LIN {X 0,Y 207.158,Z 297.304,A -85,B 0,C 180,E1 -21247.801,E2 -21247.801} C_VEL
LIN {X 0,Y 206.972,Z 297.328,A -85,B 0,C 180,E1 -21251.757,E2 -21251.757} C_VEL
LIN {X 0,Y 206.858,Z 297.342,A -85,B 0,C 180,E1 -21255.773,E2 -21255.773} C_VEL
LIN {X 0,Y 206.754,Z 297.357,A -85,B 0,C 180,E1 -21259.873,E2 -21259.873} C_VEL
LIN {X 0,Y 206.739,Z 297.359,A -85,B 0,C 180,E1 -21264.077,E2 -21264.077} C_VEL
LIN {X 0,Y 206.737,Z 297.36,A -85,B 0,C 180,E1 -21268.421,E2 -21268.421} C_VEL
LIN {X 0,Y 206.696,Z 297.365,A -85,B 0,C 180,E1 -21272.96,E2 -21272.96} C_VEL
LIN {X 0,Y 206.674,Z 297.365,A -85,B 0,C 180,E1 -21277.743,E2 -21277.743} C_VEL
LIN {X 0,Y 206.681,Z 297.525,A -85,B 0,C 180,E1 -21281.945,E2 -21281.945} C_VEL
LIN {X 0,Y 208.645,Z 305.506,A -85,B 0,C 180,E1 -21284.89,E2 -21284.89} C_VEL
LIN {X 0,Y 220.109,Z 336.47,A -85,B 0,C 180,E1 -21288.213,E2 -21288.213} C_VEL
LIN {X 0,Y 228.245,Z 359.523,A -85,B 0,C 180,E1 -21290.423,E2 -21290.423} C_VEL
LIN {X 0,Y 229.682,Z 374.179,A -85,B 0,C 180,E1 -21291.404,E2 -21291.404} C_VEL
LIN {X 0,Y 228.326,Z 390.572,A -85,B 0,C 180,E1 -21292.218,E2 -21292.218} C_VEL
LIN {X 0,Y 227.153,Z 396.303,A -85,B 0,C 180,E1 -21292.446,E2 -21292.446} C_VEL
LIN {X 0,Y 220.012,Z 414.729,A -85,B 0,C 180,E1 -21292.938,E2 -21292.938} C_VEL
LIN {X 0,Y 218.987,Z 420.451,A -85,B 0,C 180,E1 -21293.201,E2 -21293.201} C_VEL
LIN {X 0,Y 214.613,Z 474.032,A -85,B 0,C 180,E1 -21296.175,E2 -21296.175} C_VEL
LIN {X 0,Y 212.662,Z 491.06,A -85,B 0,C 180,E1 -21297.522,E2 -21297.522} C_VEL
LIN {X 0,Y 210.558,Z 506.466,A -85,B 0,C 180,E1 -21299.127,E2 -21299.127} C_VEL
LIN {X 0,Y 208.315,Z 521.44,A -85,B 0,C 180,E1 -21301.1,E2 -21301.1} C_VEL
LIN {X 0,Y 206.004,Z 535.63,A -85,B 0,C 180,E1 -21303.417,E2 -21303.417} C_VEL
LIN {X 0,Y 203.771,Z 548.988,A -85,B 0,C 180,E1 -21306.096,E2 -21306.096} C_VEL
LIN {X 0,Y 201.836,Z 561.263,A -85,B 0,C 180,E1 -21309.093,E2 -21309.093} C_VEL
LIN {X 0,Y 200.331,Z 571.626,A -85,B 0,C 180,E1 -21312.127,E2 -21312.127} C_VEL
LIN {X 0,Y 199.419,Z 580.458,A -85,B 0,C 180,E1 -21315.199,E2 -21315.199} C_VEL
LIN {X 0,Y 198.7,Z 588.985,A -85,B 0,C 180,E1 -21318.785,E2 -21318.785} C_VEL
LIN {X 0,Y 198.481,Z 596.184,A -85,B 0,C 180,E1 -21322.509,E2 -21322.509} C_VEL
LIN {X 0,Y 198.444,Z 601.423,A -85,B 0,C 180,E1 -21325.941,E2 -21325.941} C_VEL
LIN {X 0,Y 198.502,Z 605.151,A -85,B 0,C 180,E1 -21328.988,E2 -21328.988} C_VEL
LIN {X 0,Y 198.526,Z 606.143,A -85,B 0,C 180,E1 -21330.003,E2 -21330.003} C_VEL
LIN {X 0,Y 198.212,Z 607.857,A -85,B 0,C 180,E1 -21332.035,E2 -21332.035} C_VEL
LIN {X 0,Y 197.765,Z 610.327,A -85,B 0,C 180,E1 -21336.123,E2 -21336.123} C_VEL
LIN {X 0,Y 197.734,Z 611.551,A -85,B 0,C 180,E1 -21340.239,E2 -21340.239} C_VEL
LIN {X 0,Y 198.647,Z 611.744,A -85,B 0,C 180,E1 -21344.342,E2 -21344.342} C_VEL
LIN {X 0,Y 200.632,Z 610.973,A -85,B 0,C 180,E1 -21348.379,E2 -21348.379} C_VEL
LIN {X 0,Y 203.669,Z 609.172,A -85,B 0,C 180,E1 -21352.31,E2 -21352.31} C_VEL
LIN {X 0,Y 207.814,Z 606.493,A -85,B 0,C 180,E1 -21356.084,E2 -21356.084} C_VEL
LIN {X 0,Y 214.254,Z 601.836,A -85,B 0,C 180,E1 -21360.562,E2 -21360.562} C_VEL
LIN {X 0,Y 220.807,Z 596.991,A -85,B 0,C 180,E1 -21363.851,E2 -21363.851} C_VEL
LIN {X 0,Y 228.188,Z 591.239,A -85,B 0,C 180,E1 -21366.914,E2 -21366.914} C_VEL
LIN {X 0,Y 238.692,Z 582.613,A -85,B 0,C 180,E1 -21370.376,E2 -21370.376} C_VEL
LIN {X 0,Y 249.274,Z 573.413,A -85,B 0,C 180,E1 -21373.136,E2 -21373.136} C_VEL
LIN {X 0,Y 261.094,Z 562.414,A -85,B 0,C 180,E1 -21375.618,E2 -21375.618} C_VEL
LIN {X 0,Y 263.542,Z 560.056,A -85,B 0,C 180,E1 -21376.059,E2 -21376.059} C_VEL
LIN {X 0,Y 265.367,Z 558.242,A -85,B 0,C 180,E1 -21376.481,E2 -21376.481} C_VEL
LIN {X 0,Y 255.351,Z 566.825,A -85,B 0,C 180,E1 -21378.657,E2 -21378.657} C_VEL
LIN {X 0,Y 245.952,Z 574.157,A -85,B 0,C 180,E1 -21381.049,E2 -21381.049} C_VEL
LIN {X 0,Y 237.326,Z 580.309,A -85,B 0,C 180,E1 -21383.681,E2 -21383.681} C_VEL
LIN {X 0,Y 227.68,Z 586.472,A -85,B 0,C 180,E1 -21387.302,E2 -21387.302} C_VEL
LIN {X 0,Y 222.472,Z 589.437,A -85,B 0,C 180,E1 -21389.638,E2 -21389.638} C_VEL
LIN {X 0,Y 216.068,Z 592.504,A -85,B 0,C 180,E1 -21392.91,E2 -21392.91} C_VEL
LIN {X 0,Y 210.835,Z 594.559,A -85,B 0,C 180,E1 -21396.42,E2 -21396.42} C_VEL
LIN {X 0,Y 206.404,Z 595.676,A -85,B 0,C 180,E1 -21400.091,E2 -21400.091} C_VEL
LIN {X 0,Y 203.089,Z 595.732,A -85,B 0,C 180,E1 -21403.927,E2 -21403.927} C_VEL
LIN {X 0,Y 200.56,Z 594.829,A -85,B 0,C 180,E1 -21407.861,E2 -21407.861} C_VEL
LIN {X 0,Y 198.829,Z 592.903,A -85,B 0,C 180,E1 -21411.87,E2 -21411.87} C_VEL
LIN {X 0,Y 198.003,Z 589.825,A -85,B 0,C 180,E1 -21415.928,E2 -21415.928} C_VEL
LIN {X 0,Y 197.683,Z 585.567,A -85,B 0,C 180,E1 -21419.998,E2 -21419.998} C_VEL
LIN {X 0,Y 197.617,Z 579.966,A -85,B 0,C 180,E1 -21424.077,E2 -21424.077} C_VEL
LIN {X 0,Y 197.923,Z 573.55,A -85,B 0,C 180,E1 -21427.797,E2 -21427.797} C_VEL
LIN {X 0,Y 198.486,Z 566.37,A -85,B 0,C 180,E1 -21431.228,E2 -21431.228} C_VEL
LIN {X 0,Y 199.601,Z 557.396,A -85,B 0,C 180,E1 -21434.788,E2 -21434.788} C_VEL
LIN {X 0,Y 200.789,Z 548.246,A -85,B 0,C 180,E1 -21437.833,E2 -21437.833} C_VEL
LIN {X 0,Y 202.424,Z 537.538,A -85,B 0,C 180,E1 -21440.845,E2 -21440.845} C_VEL
LIN {X 0,Y 204.502,Z 524.907,A -85,B 0,C 180,E1 -21443.814,E2 -21443.814} C_VEL
LIN {X 0,Y 206.675,Z 511.004,A -85,B 0,C 180,E1 -21446.506,E2 -21446.506} C_VEL
LIN {X 0,Y 208.856,Z 497.334,A -85,B 0,C 180,E1 -21448.687,E2 -21448.687} C_VEL
LIN {X 0,Y 211.125,Z 481.108,A -85,B 0,C 180,E1 -21450.782,E2 -21450.782} C_VEL
LIN {X 0,Y 213.067,Z 465.042,A -85,B 0,C 180,E1 -21452.41,E2 -21452.41} C_VEL
LIN {X 0,Y 214.706,Z 447.806,A -85,B 0,C 180,E1 -21453.739,E2 -21453.739} C_VEL
LIN {X 0,Y 222.683,Z 352.368,A -85,B 0,C 180,E1 -21458.818,E2 -21458.818} C_VEL
LIN {X 0,Y 208.46,Z 318.723,A -85,B 0,C 180,E1 -21462.477,E2 -21462.477} C_VEL
LIN {X 0,Y 199.665,Z 298.693,A -85,B 0,C 180,E1 -21464.953,E2 -21464.953} C_VEL
LIN {X 0,Y 199.596,Z 298.249,A -85,B 0,C 180,E1 -21465.082,E2 -21465.082} C_VEL
LIN {X 0,Y 199.58,Z 298.249,A -85,B 0,C 180,E1 -21468.002,E2 -21468.002} C_VEL
LIN {X 0,Y 199.61,Z 298.243,A -85,B 0,C 180,E1 -21470.765,E2 -21470.765} C_VEL
LIN {X 0,Y 199.61,Z 298.247,A -85,B 0,C 180,E1 -21475.71,E2 -21475.71} C_VEL
LIN {X 0,Y 199.684,Z 298.235,A -85,B 0,C 180,E1 -21478.131,E2 -21478.131} C_VEL
LIN {X 0,Y 199.641,Z 298.24,A -85,B 0,C 180,E1 -21482.762,E2 -21482.762} C_VEL
LIN {X 0,Y 199.703,Z 298.233,A -85,B 0,C 180,E1 -21487.222,E2 -21487.222} C_VEL
LIN {X 0,Y 199.746,Z 298.23,A -85,B 0,C 180,E1 -21491.796,E2 -21491.796} C_VEL
LIN {X 0,Y 199.813,Z 298.223,A -85,B 0,C 180,E1 -21495.744,E2 -21495.744} C_VEL
LIN {X 0,Y 200.066,Z 298.192,A -85,B 0,C 180,E1 -21499.881,E2 -21499.881} C_VEL
LIN {X 0,Y 200.028,Z 298.192,A -85,B 0,C 180,E1 -21503.947,E2 -21503.947} C_VEL
LIN {X 0,Y 200.315,Z 298.158,A -85,B 0,C 180,E1 -21507.987,E2 -21507.987} C_VEL
LIN {X 0,Y 200.473,Z 298.136,A -85,B 0,C 180,E1 -21509.997,E2 -21509.997} C_VEL
LIN {X 0,Y 200.023,Z 298.193,A -85,B 0,C 180,E1 -21514.027,E2 -21514.027} C_VEL
LIN {X 0,Y 200.112,Z 298.181,A -85,B 0,C 180,E1 -21518.073,E2 -21518.073} C_VEL
LIN {X 0,Y 199.878,Z 298.21,A -85,B 0,C 180,E1 -21522.176,E2 -21522.176} C_VEL
LIN {X 0,Y 199.796,Z 298.22,A -85,B 0,C 180,E1 -21526.341,E2 -21526.341} C_VEL
LIN {X 0,Y 199.691,Z 298.233,A -85,B 0,C 180,E1 -21530.603,E2 -21530.603} C_VEL
LIN {X 0,Y 199.663,Z 298.238,A -85,B 0,C 180,E1 -21534.982,E2 -21534.982} C_VEL
LIN {X 0,Y 199.654,Z 298.241,A -85,B 0,C 180,E1 -21539.522,E2 -21539.522} C_VEL
LIN {X 0,Y 199.646,Z 298.239,A -85,B 0,C 180,E1 -21542.348,E2 -21542.348} C_VEL
LIN {X 0,Y 199.628,Z 298.24,A -85,B 0,C 180,E1 -21546.758,E2 -21546.758} C_VEL
LIN {X 0,Y 199.626,Z 298.245,A -85,B 0,C 180,E1 -21549.32,E2 -21549.32} C_VEL
LIN {X 0,Y 199.568,Z 298.246,A -85,B 0,C 180,E1 -21554.77,E2 -21554.77} C_VEL
LIN {X 0,Y 199.567,Z 298.25,A -85,B 0,C 180,E1 -21558.004,E2 -21558.004} C_VEL
LIN {X 0,Y 199.598,Z 298.245,A -85,B 0,C 180,E1 -21560.767,E2 -21560.767} C_VEL
LIN {X 0,Y 199.601,Z 298.246,A -85,B 0,C 180,E1 -21565.714,E2 -21565.714} C_VEL
LIN {X 0,Y 199.688,Z 298.234,A -85,B 0,C 180,E1 -21568.137,E2 -21568.137} C_VEL
LIN {X 0,Y 199.674,Z 298.235,A -85,B 0,C 180,E1 -21572.772,E2 -21572.772} C_VEL
LIN {X 0,Y 199.702,Z 298.233,A -85,B 0,C 180,E1 -21577.227,E2 -21577.227} C_VEL
LIN {X 0,Y 199.784,Z 298.222,A -85,B 0,C 180,E1 -21581.759,E2 -21581.759} C_VEL
LIN {X 0,Y 199.836,Z 298.215,A -85,B 0,C 180,E1 -21585.75,E2 -21585.75} C_VEL
LIN {X 0,Y 200.059,Z 298.187,A -85,B 0,C 180,E1 -21589.885,E2 -21589.885} C_VEL
LIN {X 0,Y 200.022,Z 298.192,A -85,B 0,C 180,E1 -21593.951,E2 -21593.951} C_VEL
LIN {X 0,Y 200.31,Z 298.156,A -85,B 0,C 180,E1 -21597.991,E2 -21597.991} C_VEL
LIN {X 0,Y 200.468,Z 298.137,A -85,B 0,C 180,E1 -21600.002,E2 -21600.002} C_VEL
LIN {X 0,Y 200.018,Z 298.193,A -85,B 0,C 180,E1 -21604.031,E2 -21604.031} C_VEL
LIN {X 0,Y 200.102,Z 298.183,A -85,B 0,C 180,E1 -21608.078,E2 -21608.078} C_VEL
LIN {X 0,Y 199.904,Z 298.208,A -85,B 0,C 180,E1 -21612.179,E2 -21612.179} C_VEL
LIN {X 0,Y 199.795,Z 298.223,A -85,B 0,C 180,E1 -21616.346,E2 -21616.346} C_VEL
LIN {X 0,Y 199.673,Z 298.241,A -85,B 0,C 180,E1 -21620.61,E2 -21620.61} C_VEL
LIN {X 0,Y 199.657,Z 298.244,A -85,B 0,C 180,E1 -21624.988,E2 -21624.988} C_VEL
LIN {X 0,Y 199.668,Z 298.239,A -85,B 0,C 180,E1 -21629.525,E2 -21629.525} C_VEL
LIN {X 0,Y 199.671,Z 298.239,A -85,B 0,C 180,E1 -21632.361,E2 -21632.361} C_VEL
LIN {X 0,Y 199.617,Z 298.246,A -85,B 0,C 180,E1 -21636.766,E2 -21636.766} C_VEL
LIN {X 0,Y 199.643,Z 298.323,A -85,B 0,C 180,E1 -21641.306,E2 -21641.306} C_VEL
LIN {X 0,Y 201.172,Z 304.852,A -85,B 0,C 180,E1 -21643.849,E2 -21643.849} C_VEL
LIN {X 0,Y 211.896,Z 333.808,A -85,B 0,C 180,E1 -21647.122,E2 -21647.122} C_VEL
LIN {X 0,Y 221.672,Z 361.387,A -85,B 0,C 180,E1 -21649.884,E2 -21649.884} C_VEL
LIN {X 0,Y 222.987,Z 374.723,A -85,B 0,C 180,E1 -21650.81,E2 -21650.81} C_VEL
LIN {X 0,Y 218.987,Z 420.451,A -85,B 0,C 180,E1 -21653.201,E2 -21653.201} C_VEL
LIN {X 0,Y 217.932,Z 426.174,A -85,B 0,C 180,E1 -21653.459,E2 -21653.459} C_VEL
LIN {X 0,Y 210.751,Z 444.563,A -85,B 0,C 180,E1 -21654.048,E2 -21654.048} C_VEL
LIN {X 0,Y 209.668,Z 450.283,A -85,B 0,C 180,E1 -21654.333,E2 -21654.333} C_VEL
LIN {X 0,Y 207.486,Z 475.638,A -85,B 0,C 180,E1 -21655.878,E2 -21655.878} C_VEL
LIN {X 0,Y 205.561,Z 492.17,A -85,B 0,C 180,E1 -21657.278,E2 -21657.278} C_VEL
LIN {X 0,Y 203.262,Z 508.372,A -85,B 0,C 180,E1 -21659.081,E2 -21659.081} C_VEL
LIN {X 0,Y 200.895,Z 523.396,A -85,B 0,C 180,E1 -21661.211,E2 -21661.211} C_VEL
LIN {X 0,Y 198.522,Z 537.713,A -85,B 0,C 180,E1 -21663.739,E2 -21663.739} C_VEL
LIN {X 0,Y 196.331,Z 550.691,A -85,B 0,C 180,E1 -21666.535,E2 -21666.535} C_VEL
LIN {X 0,Y 194.422,Z 563.417,A -85,B 0,C 180,E1 -21669.883,E2 -21669.883} C_VEL
LIN {X 0,Y 192.977,Z 573.41,A -85,B 0,C 180,E1 -21673.064,E2 -21673.064} C_VEL
LIN {X 0,Y 192.145,Z 581.857,A -85,B 0,C 180,E1 -21676.25,E2 -21676.25} C_VEL
LIN {X 0,Y 191.613,Z 590.021,A -85,B 0,C 180,E1 -21679.97,E2 -21679.97} C_VEL
LIN {X 0,Y 191.521,Z 596.662,A -85,B 0,C 180,E1 -21683.683,E2 -21683.683} C_VEL
LIN {X 0,Y 191.482,Z 601.152,A -85,B 0,C 180,E1 -21686.847,E2 -21686.847} C_VEL
LIN {X 0,Y 191.545,Z 604.766,A -85,B 0,C 180,E1 -21690.003,E2 -21690.003} C_VEL
LIN {X 0,Y 191.218,Z 606.595,A -85,B 0,C 180,E1 -21692.109,E2 -21692.109} C_VEL
LIN {X 0,Y 190.763,Z 609.227,A -85,B 0,C 180,E1 -21696.348,E2 -21696.348} C_VEL
LIN {X 0,Y 190.731,Z 610.696,A -85,B 0,C 180,E1 -21700.62,E2 -21700.62} C_VEL
LIN {X 0,Y 191.737,Z 611.159,A -85,B 0,C 180,E1 -21704.87,E2 -21704.87} C_VEL
LIN {X 0,Y 194.399,Z 610.364,A -85,B 0,C 180,E1 -21709.951,E2 -21709.951} C_VEL
LIN {X 0,Y 197.07,Z 609.151,A -85,B 0,C 180,E1 -21713.1,E2 -21713.1} C_VEL
LIN {X 0,Y 201.44,Z 606.724,A -85,B 0,C 180,E1 -21716.975,E2 -21716.975} C_VEL
LIN {X 0,Y 206.711,Z 603.475,A -85,B 0,C 180,E1 -21720.666,E2 -21720.666} C_VEL
LIN {X 0,Y 211.433,Z 600.418,A -85,B 0,C 180,E1 -21723.264,E2 -21723.264} C_VEL
LIN {X 0,Y 220.692,Z 594.186,A -85,B 0,C 180,E1 -21727.236,E2 -21727.236} C_VEL
LIN {X 0,Y 229.057,Z 588.162,A -85,B 0,C 180,E1 -21730.118,E2 -21730.118} C_VEL
LIN {X 0,Y 238.246,Z 581.142,A -85,B 0,C 180,E1 -21732.727,E2 -21732.727} C_VEL
LIN {X 0,Y 249.598,Z 571.963,A -85,B 0,C 180,E1 -21735.317,E2 -21735.317} C_VEL
LIN {X 0,Y 255.701,Z 566.726,A -85,B 0,C 180,E1 -21736.595,E2 -21736.595} C_VEL
LIN {X 0,Y 245.688,Z 574.093,A -85,B 0,C 180,E1 -21738.857,E2 -21738.857} C_VEL
LIN {X 0,Y 236.392,Z 580.304,A -85,B 0,C 180,E1 -21741.365,E2 -21741.365} C_VEL
LIN {X 0,Y 227.884,Z 585.449,A -85,B 0,C 180,E1 -21744.128,E2 -21744.128} C_VEL
LIN {X 0,Y 220.154,Z 589.537,A -85,B 0,C 180,E1 -21747.132,E2 -21747.132} C_VEL
LIN {X 0,Y 213.232,Z 592.706,A -85,B 0,C 180,E1 -21750.369,E2 -21750.369} C_VEL
LIN {X 0,Y 209.911,Z 593.986,A -85,B 0,C 180,E1 -21752.047,E2 -21752.047} C_VEL
LIN {X 0,Y 204.422,Z 595.675,A -85,B 0,C 180,E1 -21755.633,E2 -21755.633} C_VEL
LIN {X 0,Y 199.796,Z 596.434,A -85,B 0,C 180,E1 -21759.404,E2 -21759.404} C_VEL
LIN {X 0,Y 196.273,Z 596.26,A -85,B 0,C 180,E1 -21763.352,E2 -21763.352} C_VEL
LIN {X 0,Y 193.642,Z 595.035,A -85,B 0,C 180,E1 -21767.421,E2 -21767.421} C_VEL
LIN {X 0,Y 191.741,Z 592.67,A -85,B 0,C 180,E1 -21771.764,E2 -21771.764} C_VEL
LIN {X 0,Y 190.833,Z 588.472,A -85,B 0,C 180,E1 -21776.832,E2 -21776.832} C_VEL
LIN {X 0,Y 190.583,Z 583.629,A -85,B 0,C 180,E1 -21781.055,E2 -21781.055} C_VEL
LIN {X 0,Y 190.595,Z 578.073,A -85,B 0,C 180,E1 -21784.872,E2 -21784.872} C_VEL
LIN {X 0,Y 191.061,Z 570.604,A -85,B 0,C 180,E1 -21788.992,E2 -21788.992} C_VEL
LIN {X 0,Y 191.803,Z 562.401,A -85,B 0,C 180,E1 -21792.698,E2 -21792.698} C_VEL
LIN {X 0,Y 193.105,Z 552.548,A -85,B 0,C 180,E1 -21796.381,E2 -21796.381} C_VEL
LIN {X 0,Y 194.549,Z 542.52,A -85,B 0,C 180,E1 -21799.532,E2 -21799.532} C_VEL
LIN {X 0,Y 196.39,Z 530.744,A -85,B 0,C 180,E1 -21802.623,E2 -21802.623} C_VEL
LIN {X 0,Y 198.514,Z 517.98,A -85,B 0,C 180,E1 -21805.419,E2 -21805.419} C_VEL
LIN {X 0,Y 200.748,Z 504.22,A -85,B 0,C 180,E1 -21807.918,E2 -21807.918} C_VEL
LIN {X 0,Y 202.993,Z 489.35,A -85,B 0,C 180,E1 -21810.122,E2 -21810.122} C_VEL
LIN {X 0,Y 205.235,Z 472.959,A -85,B 0,C 180,E1 -21812.056,E2 -21812.056} C_VEL
LIN {X 0,Y 207.087,Z 455.951,A -85,B 0,C 180,E1 -21813.612,E2 -21813.612} C_VEL
LIN {X 0,Y 208.745,Z 437.25,A -85,B 0,C 180,E1 -21814.839,E2 -21814.839} C_VEL
LIN {X 0,Y 215.881,Z 353.963,A -85,B 0,C 180,E1 -21819.405,E2 -21819.405} C_VEL
LIN {X 0,Y 202.549,Z 322.266,A -85,B 0,C 180,E1 -21822.963,E2 -21822.963} C_VEL
LIN {X 0,Y 192.658,Z 299.933,A -85,B 0,C 180,E1 -21825.848,E2 -21825.848} C_VEL
LIN {X 0,Y 192.497,Z 299.133,A -85,B 0,C 180,E1 -21825.983,E2 -21825.983} C_VEL
LIN {X 0,Y 192.518,Z 299.128,A -85,B 0,C 180,E1 -21830.048,E2 -21830.048} C_VEL
LIN {X 0,Y 192.56,Z 299.122,A -85,B 0,C 180,E1 -21834.267,E2 -21834.267} C_VEL
LIN {X 0,Y 192.604,Z 299.119,A -85,B 0,C 180,E1 -21837.058,E2 -21837.058} C_VEL
LIN {X 0,Y 192.619,Z 299.118,A -85,B 0,C 180,E1 -21841.682,E2 -21841.682} C_VEL
LIN {X 0,Y 192.675,Z 299.108,A -85,B 0,C 180,E1 -21846.342,E2 -21846.342} C_VEL
LIN {X 0,Y 192.694,Z 299.109,A -85,B 0,C 180,E1 -21851.485,E2 -21851.485} C_VEL
LIN {X 0,Y 192.737,Z 299.105,A -85,B 0,C 180,E1 -21855.209,E2 -21855.209} C_VEL
LIN {X 0,Y 192.977,Z 299.075,A -85,B 0,C 180,E1 -21859.505,E2 -21859.505} C_VEL
LIN {X 0,Y 193.057,Z 299.065,A -85,B 0,C 180,E1 -21861.624,E2 -21861.624} C_VEL
LIN {X 0,Y 193.257,Z 299.038,A -85,B 0,C 180,E1 -21867.913,E2 -21867.913} C_VEL
LIN {X 0,Y 193.437,Z 299.012,A -85,B 0,C 180,E1 -21869.997,E2 -21869.997} C_VEL
LIN {X 0,Y 192.97,Z 299.071,A -85,B 0,C 180,E1 -21874.174,E2 -21874.174} C_VEL
LIN {X 0,Y 193.061,Z 299.058,A -85,B 0,C 180,E1 -21878.37,E2 -21878.37} C_VEL
LIN {X 0,Y 192.802,Z 299.091,A -85,B 0,C 180,E1 -21882.63,E2 -21882.63} C_VEL
LIN {X 0,Y 192.749,Z 299.099,A -85,B 0,C 180,E1 -21886.956,E2 -21886.956} C_VEL
LIN {X 0,Y 192.627,Z 299.116,A -85,B 0,C 180,E1 -21891.395,E2 -21891.395} C_VEL
LIN {X 0,Y 192.654,Z 299.11,A -85,B 0,C 180,E1 -21894.222,E2 -21894.222} C_VEL
LIN {X 0,Y 192.633,Z 299.112,A -85,B 0,C 180,E1 -21898.887,E2 -21898.887} C_VEL
LIN {X 0,Y 192.587,Z 299.121,A -85,B 0,C 180,E1 -21903.184,E2 -21903.184} C_VEL
LIN {X 0,Y 192.562,Z 299.122,A -85,B 0,C 180,E1 -21908.345,E2 -21908.345} C_VEL
LIN {X 0,Y 192.48,Z 299.132,A -85,B 0,C 180,E1 -21913.095,E2 -21913.095} C_VEL
LIN {X 0,Y 192.479,Z 299.133,A -85,B 0,C 180,E1 -21916.903,E2 -21916.903} C_VEL
LIN {X 0,Y 192.539,Z 299.122,A -85,B 0,C 180,E1 -21921.648,E2 -21921.648} C_VEL
LIN {X 0,Y 192.586,Z 299.12,A -85,B 0,C 180,E1 -21926.814,E2 -21926.814} C_VEL
LIN {X 0,Y 192.652,Z 299.11,A -85,B 0,C 180,E1 -21931.692,E2 -21931.692} C_VEL
LIN {X 0,Y 192.673,Z 299.108,A -85,B 0,C 180,E1 -21936.346,E2 -21936.346} C_VEL
LIN {X 0,Y 192.719,Z 299.104,A -85,B 0,C 180,E1 -21941.459,E2 -21941.459} C_VEL
LIN {X 0,Y 192.76,Z 299.098,A -85,B 0,C 180,E1 -21945.215,E2 -21945.215} C_VEL
LIN {X 0,Y 192.97,Z 299.072,A -85,B 0,C 180,E1 -21949.51,E2 -21949.51} C_VEL
LIN {X 0,Y 193.05,Z 299.062,A -85,B 0,C 180,E1 -21951.629,E2 -21951.629} C_VEL
LIN {X 0,Y 193.252,Z 299.035,A -85,B 0,C 180,E1 -21957.918,E2 -21957.918} C_VEL
LIN {X 0,Y 193.432,Z 299.013,A -85,B 0,C 180,E1 -21960.002,E2 -21960.002} C_VEL
LIN {X 0,Y 192.965,Z 299.071,A -85,B 0,C 180,E1 -21964.179,E2 -21964.179} C_VEL
LIN {X 0,Y 193.052,Z 299.061,A -85,B 0,C 180,E1 -21968.375,E2 -21968.375} C_VEL
LIN {X 0,Y 192.843,Z 299.089,A -85,B 0,C 180,E1 -21972.632,E2 -21972.632} C_VEL
LIN {X 0,Y 192.748,Z 299.103,A -85,B 0,C 180,E1 -21976.961,E2 -21976.961} C_VEL
LIN {X 0,Y 192.608,Z 299.12,A -85,B 0,C 180,E1 -21981.402,E2 -21981.402} C_VEL
LIN {X 0,Y 192.639,Z 299.116,A -85,B 0,C 180,E1 -21984.216,E2 -21984.216} C_VEL
LIN {X 0,Y 192.643,Z 299.118,A -85,B 0,C 180,E1 -21988.895,E2 -21988.895} C_VEL
LIN {X 0,Y 192.592,Z 299.121,A -85,B 0,C 180,E1 -21993.189,E2 -21993.189} C_VEL
LIN {X 0,Y 192.545,Z 299.126,A -85,B 0,C 180,E1 -21998.355,E2 -21998.355} C_VEL
LIN {X 0,Y 192.605,Z 299.17,A -85,B 0,C 180,E1 -22000.657,E2 -22000.657} C_VEL
LIN {X 0,Y 193.869,Z 304.631,A -85,B 0,C 180,E1 -22002.823,E2 -22002.823} C_VEL
LIN {X 0,Y 204.056,Z 332.015,A -85,B 0,C 180,E1 -22006.074,E2 -22006.074} C_VEL
LIN {X 0,Y 214.809,Z 362.468,A -85,B 0,C 180,E1 -22009.256,E2 -22009.256} C_VEL
LIN {X 0,Y 215.795,Z 369.657,A -85,B 0,C 180,E1 -22009.804,E2 -22009.804} C_VEL
LIN {X 0,Y 216.24,Z 375.682,A -85,B 0,C 180,E1 -22010.222,E2 -22010.222} C_VEL
LIN {X 0,Y 209.668,Z 450.283,A -85,B 0,C 180,E1 -22014.333,E2 -22014.333} C_VEL
LIN {X 0,Y 208.721,Z 454.098,A -85,B 0,C 180,E1 -22014.507,E2 -22014.507} C_VEL
LIN {X 0,Y 202.146,Z 465.851,A -85,B 0,C 180,E1 -22014.835,E2 -22014.835} C_VEL
LIN {X 0,Y 201.179,Z 469.651,A -85,B 0,C 180,E1 -22015.044,E2 -22015.044} C_VEL
LIN {X 0,Y 199.213,Z 486.792,A -85,B 0,C 180,E1 -22016.401,E2 -22016.401} C_VEL
LIN {X 0,Y 197.18,Z 501.788,A -85,B 0,C 180,E1 -22017.986,E2 -22017.986} C_VEL
LIN {X 0,Y 194.829,Z 516.94,A -85,B 0,C 180,E1 -22020.028,E2 -22020.028} C_VEL
LIN {X 0,Y 192.369,Z 531.804,A -85,B 0,C 180,E1 -22022.536,E2 -22022.536} C_VEL
LIN {X 0,Y 190.008,Z 545.642,A -85,B 0,C 180,E1 -22025.414,E2 -22025.414} C_VEL
LIN {X 0,Y 187.975,Z 558.169,A -85,B 0,C 180,E1 -22028.587,E2 -22028.587} C_VEL
LIN {X 0,Y 186.391,Z 568.887,A -85,B 0,C 180,E1 -22031.88,E2 -22031.88} C_VEL
LIN {X 0,Y 185.452,Z 577.917,A -85,B 0,C 180,E1 -22035.182,E2 -22035.182} C_VEL
LIN {X 0,Y 184.749,Z 586.682,A -85,B 0,C 180,E1 -22039.038,E2 -22039.038} C_VEL
LIN {X 0,Y 184.562,Z 593.686,A -85,B 0,C 180,E1 -22042.822,E2 -22042.822} C_VEL
LIN {X 0,Y 184.524,Z 597.988,A -85,B 0,C 180,E1 -22045.634,E2 -22045.634} C_VEL
LIN {X 0,Y 184.595,Z 602.093,A -85,B 0,C 180,E1 -22048.912,E2 -22048.912} C_VEL
LIN {X 0,Y 184.62,Z 603.236,A -85,B 0,C 180,E1 -22050.003,E2 -22050.003} C_VEL
LIN {X 0,Y 184.255,Z 605.179,A -85,B 0,C 180,E1 -22052.189,E2 -22052.189} C_VEL
LIN {X 0,Y 183.773,Z 608.077,A -85,B 0,C 180,E1 -22056.591,E2 -22056.591} C_VEL
LIN {X 0,Y 183.745,Z 609.775,A -85,B 0,C 180,E1 -22061.028,E2 -22061.028} C_VEL
LIN {X 0,Y 184.847,Z 610.442,A -85,B 0,C 180,E1 -22065.438,E2 -22065.438} C_VEL
LIN {X 0,Y 187.473,Z 610.062,A -85,B 0,C 180,E1 -22070.41,E2 -22070.41} C_VEL
LIN {X 0,Y 192.688,Z 608.062,A -85,B 0,C 180,E1 -22075.959,E2 -22075.959} C_VEL
LIN {X 0,Y 197.73,Z 605.56,A -85,B 0,C 180,E1 -22079.845,E2 -22079.845} C_VEL
LIN {X 0,Y 203.831,Z 602.201,A -85,B 0,C 180,E1 -22083.485,E2 -22083.485} C_VEL
LIN {X 0,Y 213.162,Z 596.772,A -85,B 0,C 180,E1 -22087.589,E2 -22087.589} C_VEL
LIN {X 0,Y 223.855,Z 589.959,A -85,B 0,C 180,E1 -22091.249,E2 -22091.249} C_VEL
LIN {X 0,Y 233.314,Z 583.475,A -85,B 0,C 180,E1 -22093.856,E2 -22093.856} C_VEL
LIN {X 0,Y 245.937,Z 574.201,A -85,B 0,C 180,E1 -22096.697,E2 -22096.697} C_VEL
LIN {X 0,Y 235.974,Z 580.465,A -85,B 0,C 180,E1 -22099.062,E2 -22099.062} C_VEL
LIN {X 0,Y 224.604,Z 586.746,A -85,B 0,C 180,E1 -22102.397,E2 -22102.397} C_VEL
LIN {X 0,Y 214.462,Z 591.504,A -85,B 0,C 180,E1 -22106.143,E2 -22106.143} C_VEL
LIN {X 0,Y 207.259,Z 594.275,A -85,B 0,C 180,E1 -22109.425,E2 -22109.425} C_VEL
LIN {X 0,Y 203.799,Z 595.341,A -85,B 0,C 180,E1 -22111.131,E2 -22111.131} C_VEL
LIN {X 0,Y 198.045,Z 596.708,A -85,B 0,C 180,E1 -22114.794,E2 -22114.794} C_VEL
LIN {X 0,Y 193.221,Z 597.169,A -85,B 0,C 180,E1 -22118.669,E2 -22118.669} C_VEL
LIN {X 0,Y 189.488,Z 596.63,A -85,B 0,C 180,E1 -22122.738,E2 -22122.738} C_VEL
LIN {X 0,Y 186.719,Z 595.162,A -85,B 0,C 180,E1 -22126.946,E2 -22126.946} C_VEL
LIN {X 0,Y 184.602,Z 592.237,A -85,B 0,C 180,E1 -22131.845,E2 -22131.845} C_VEL
LIN {X 0,Y 183.78,Z 588.006,A -85,B 0,C 180,E1 -22136.71,E2 -22136.71} C_VEL
LIN {X 0,Y 183.519,Z 582.88,A -85,B 0,C 180,E1 -22141.095,E2 -22141.095} C_VEL
LIN {X 0,Y 183.587,Z 576.269,A -85,B 0,C 180,E1 -22145.519,E2 -22145.519} C_VEL
LIN {X 0,Y 184.124,Z 568.123,A -85,B 0,C 180,E1 -22149.889,E2 -22149.889} C_VEL
LIN {X 0,Y 185.045,Z 559.329,A -85,B 0,C 180,E1 -22153.73,E2 -22153.73} C_VEL
LIN {X 0,Y 186.287,Z 550.435,A -85,B 0,C 180,E1 -22156.999,E2 -22156.999} C_VEL
LIN {X 0,Y 187.992,Z 538.822,A -85,B 0,C 180,E1 -22160.582,E2 -22160.582} C_VEL
LIN {X 0,Y 190.003,Z 526.594,A -85,B 0,C 180,E1 -22163.717,E2 -22163.717} C_VEL
LIN {X 0,Y 192.232,Z 513.045,A -85,B 0,C 180,E1 -22166.604,E2 -22166.604} C_VEL
LIN {X 0,Y 194.684,Z 498.235,A -85,B 0,C 180,E1 -22169.164,E2 -22169.164} C_VEL
LIN {X 0,Y 196.875,Z 482.974,A -85,B 0,C 180,E1 -22171.302,E2 -22171.302} C_VEL
LIN {X 0,Y 198.915,Z 467.252,A -85,B 0,C 180,E1 -22173.052,E2 -22173.052} C_VEL
LIN {X 0,Y 200.724,Z 450.033,A -85,B 0,C 180,E1 -22174.523,E2 -22174.523} C_VEL
LIN {X 0,Y 203.799,Z 413.596,A -85,B 0,C 180,E1 -22176.732,E2 -22176.732} C_VEL
LIN {X 0,Y 209.139,Z 356.299,A -85,B 0,C 180,E1 -22179.959,E2 -22179.959} C_VEL
LIN {X 0,Y 207.4,Z 351.527,A -85,B 0,C 180,E1 -22180.449,E2 -22180.449} C_VEL
LIN {X 0,Y 196.329,Z 325.13,A -85,B 0,C 180,E1 -22183.537,E2 -22183.537} C_VEL
LIN {X 0,Y 186.125,Z 302.228,A -85,B 0,C 180,E1 -22186.617,E2 -22186.617} C_VEL
LIN {X 0,Y 185.471,Z 300.008,A -85,B 0,C 180,E1 -22186.897,E2 -22186.897} C_VEL
LIN {X 0,Y 185.468,Z 300.007,A -85,B 0,C 180,E1 -22189.892,E2 -22189.892} C_VEL
LIN {X 0,Y 185.506,Z 300.003,A -85,B 0,C 180,E1 -22192.708,E2 -22192.708} C_VEL
LIN {X 0,Y 185.53,Z 299.998,A -85,B 0,C 180,E1 -22197.969,E2 -22197.969} C_VEL
LIN {X 0,Y 185.545,Z 299.996,A -85,B 0,C 180,E1 -22200.592,E2 -22200.592} C_VEL
LIN {X 0,Y 185.578,Z 299.994,A -85,B 0,C 180,E1 -22205.378,E2 -22205.378} C_VEL
LIN {X 0,Y 185.63,Z 299.988,A -85,B 0,C 180,E1 -22211.168,E2 -22211.168} C_VEL
LIN {X 0,Y 185.666,Z 299.984,A -85,B 0,C 180,E1 -22214.632,E2 -22214.632} C_VEL
LIN {X 0,Y 185.92,Z 299.953,A -85,B 0,C 180,E1 -22219.356,E2 -22219.356} C_VEL
LIN {X 0,Y 185.955,Z 299.946,A -85,B 0,C 180,E1 -22223.487,E2 -22223.487} C_VEL
LIN {X 0,Y 186.201,Z 299.917,A -85,B 0,C 180,E1 -22227.834,E2 -22227.834} C_VEL
LIN {X 0,Y 186.4,Z 299.889,A -85,B 0,C 180,E1 -22229.997,E2 -22229.997} C_VEL
LIN {X 0,Y 185.917,Z 299.949,A -85,B 0,C 180,E1 -22234.333,E2 -22234.333} C_VEL
LIN {X 0,Y 186.006,Z 299.937,A -85,B 0,C 180,E1 -22238.69,E2 -22238.69} C_VEL
LIN {X 0,Y 185.726,Z 299.974,A -85,B 0,C 180,E1 -22243.12,E2 -22243.12} C_VEL
LIN {X 0,Y 185.681,Z 299.977,A -85,B 0,C 180,E1 -22247.622,E2 -22247.622} C_VEL
LIN {X 0,Y 185.587,Z 299.991,A -85,B 0,C 180,E1 -22252.249,E2 -22252.249} C_VEL
LIN {X 0,Y 185.55,Z 299.993,A -85,B 0,C 180,E1 -22257.03,E2 -22257.03} C_VEL
LIN {X 0,Y 185.567,Z 299.995,A -85,B 0,C 180,E1 -22259.491,E2 -22259.491} C_VEL
LIN {X 0,Y 185.498,Z 300,A -85,B 0,C 180,E1 -22264.628,E2 -22264.628} C_VEL
LIN {X 0,Y 185.532,Z 299.998,A -85,B 0,C 180,E1 -22267.303,E2 -22267.303} C_VEL
LIN {X 0,Y 185.472,Z 300.006,A -85,B 0,C 180,E1 -22270.728,E2 -22270.728} C_VEL
LIN {X 0,Y 185.449,Z 300.007,A -85,B 0,C 180,E1 -22276.054,E2 -22276.054} C_VEL
LIN {X 0,Y 185.456,Z 300.007,A -85,B 0,C 180,E1 -22279.895,E2 -22279.895} C_VEL
LIN {X 0,Y 185.493,Z 299.999,A -85,B 0,C 180,E1 -22282.711,E2 -22282.711} C_VEL
LIN {X 0,Y 185.534,Z 299.997,A -85,B 0,C 180,E1 -22287.975,E2 -22287.975} C_VEL
LIN {X 0,Y 185.57,Z 299.99,A -85,B 0,C 180,E1 -22290.576,E2 -22290.576} C_VEL
LIN {X 0,Y 185.568,Z 299.995,A -85,B 0,C 180,E1 -22295.382,E2 -22295.382} C_VEL
LIN {X 0,Y 185.661,Z 299.982,A -85,B 0,C 180,E1 -22301.135,E2 -22301.135} C_VEL
LIN {X 0,Y 185.753,Z 299.97,A -85,B 0,C 180,E1 -22306.881,E2 -22306.881} C_VEL
LIN {X 0,Y 185.997,Z 299.942,A -85,B 0,C 180,E1 -22311.309,E2 -22311.309} C_VEL
LIN {X 0,Y 186.196,Z 299.914,A -85,B 0,C 180,E1 -22317.839,E2 -22317.839} C_VEL
LIN {X 0,Y 186.396,Z 299.89,A -85,B 0,C 180,E1 -22320.002,E2 -22320.002} C_VEL
LIN {X 0,Y 185.913,Z 299.95,A -85,B 0,C 180,E1 -22324.338,E2 -22324.338} C_VEL
LIN {X 0,Y 185.999,Z 299.941,A -85,B 0,C 180,E1 -22328.695,E2 -22328.695} C_VEL
LIN {X 0,Y 185.755,Z 299.973,A -85,B 0,C 180,E1 -22333.123,E2 -22333.123} C_VEL
LIN {X 0,Y 185.665,Z 299.986,A -85,B 0,C 180,E1 -22338.868,E2 -22338.868} C_VEL
LIN {X 0,Y 185.569,Z 299.998,A -85,B 0,C 180,E1 -22344.649,E2 -22344.649} C_VEL
LIN {X 0,Y 185.572,Z 299.995,A -85,B 0,C 180,E1 -22349.496,E2 -22349.496} C_VEL
LIN {X 0,Y 185.493,Z 300.005,A -85,B 0,C 180,E1 -22354.635,E2 -22354.635} C_VEL
LIN {X 0,Y 185.535,Z 300.015,A -85,B 0,C 180,E1 -22360.001,E2 -22360.001} C_VEL
LIN {X 0,Y 186.507,Z 304.274,A -85,B 0,C 180,E1 -22361.727,E2 -22361.727} C_VEL
LIN {X 0,Y 196.486,Z 330.995,A -85,B 0,C 180,E1 -22365.06,E2 -22365.06} C_VEL
LIN {X 0,Y 208.416,Z 364.877,A -85,B 0,C 180,E1 -22368.749,E2 -22368.749} C_VEL
LIN {X 0,Y 209.558,Z 375.752,A -85,B 0,C 180,E1 -22369.573,E2 -22369.573} C_VEL
LIN {X 0,Y 201.179,Z 469.651,A -85,B 0,C 180,E1 -22375.044,E2 -22375.044} C_VEL
LIN {X 0,Y 199.996,Z 475.295,A -85,B 0,C 180,E1 -22375.404,E2 -22375.404} C_VEL
LIN {X 0,Y 196.082,Z 484.195,A -85,B 0,C 180,E1 -22375.981,E2 -22375.981} C_VEL
LIN {X 0,Y 192.009,Z 492.95,A -85,B 0,C 180,E1 -22376.7,E2 -22376.7} C_VEL
LIN {X 0,Y 190.635,Z 498.373,A -85,B 0,C 180,E1 -22377.29,E2 -22377.29} C_VEL
LIN {X 0,Y 188.151,Z 514.492,A -85,B 0,C 180,E1 -22379.449,E2 -22379.449} C_VEL
LIN {X 0,Y 185.808,Z 528.382,A -85,B 0,C 180,E1 -22381.787,E2 -22381.787} C_VEL
LIN {X 0,Y 183.569,Z 541.491,A -85,B 0,C 180,E1 -22384.491,E2 -22384.491} C_VEL
LIN {X 0,Y 181.333,Z 554.807,A -85,B 0,C 180,E1 -22387.849,E2 -22387.849} C_VEL
LIN {X 0,Y 179.71,Z 565.754,A -85,B 0,C 180,E1 -22391.181,E2 -22391.181} C_VEL
LIN {X 0,Y 178.476,Z 576.541,A -85,B 0,C 180,E1 -22395.173,E2 -22395.173} C_VEL
LIN {X 0,Y 177.8,Z 585.424,A -85,B 0,C 180,E1 -22399.181,E2 -22399.181} C_VEL
LIN {X 0,Y 177.613,Z 592.66,A -85,B 0,C 180,E1 -22403.186,E2 -22403.186} C_VEL
LIN {X 0,Y 177.593,Z 597.649,A -85,B 0,C 180,E1 -22406.6,E2 -22406.6} C_VEL
LIN {X 0,Y 177.685,Z 601.649,A -85,B 0,C 180,E1 -22410.003,E2 -22410.003} C_VEL
LIN {X 0,Y 177.301,Z 603.726,A -85,B 0,C 180,E1 -22412.275,E2 -22412.275} C_VEL
LIN {X 0,Y 176.789,Z 606.823,A -85,B 0,C 180,E1 -22416.853,E2 -22416.853} C_VEL
LIN {X 0,Y 176.816,Z 608.736,A -85,B 0,C 180,E1 -22421.466,E2 -22421.466} C_VEL
LIN {X 0,Y 177.98,Z 609.695,A -85,B 0,C 180,E1 -22426.049,E2 -22426.049} C_VEL
LIN {X 0,Y 180.58,Z 609.613,A -85,B 0,C 180,E1 -22430.92,E2 -22430.92} C_VEL
LIN {X 0,Y 184.007,Z 608.799,A -85,B 0,C 180,E1 -22434.846,E2 -22434.846} C_VEL
LIN {X 0,Y 191.589,Z 605.823,A -85,B 0,C 180,E1 -22440.904,E2 -22440.904} C_VEL
LIN {X 0,Y 197.968,Z 602.822,A -85,B 0,C 180,E1 -22444.615,E2 -22444.615} C_VEL
LIN {X 0,Y 206.943,Z 598.274,A -85,B 0,C 180,E1 -22448.486,E2 -22448.486} C_VEL
LIN {X 0,Y 216.401,Z 593.021,A -85,B 0,C 180,E1 -22451.745,E2 -22451.745} C_VEL
LIN {X 0,Y 228.447,Z 585.705,A -85,B 0,C 180,E1 -22455.041,E2 -22455.041} C_VEL
LIN {X 0,Y 236.085,Z 580.713,A -85,B 0,C 180,E1 -22456.788,E2 -22456.788} C_VEL
LIN {X 0,Y 223.902,Z 587.031,A -85,B 0,C 180,E1 -22459.948,E2 -22459.948} C_VEL
LIN {X 0,Y 212.885,Z 591.856,A -85,B 0,C 180,E1 -22463.54,E2 -22463.54} C_VEL
LIN {X 0,Y 204.955,Z 594.653,A -85,B 0,C 180,E1 -22466.724,E2 -22466.724} C_VEL
LIN {X 0,Y 197.737,Z 596.643,A -85,B 0,C 180,E1 -22470.158,E2 -22470.158} C_VEL
LIN {X 0,Y 191.714,Z 597.659,A -85,B 0,C 180,E1 -22473.901,E2 -22473.901} C_VEL
LIN {X 0,Y 186.642,Z 597.766,A -85,B 0,C 180,E1 -22477.878,E2 -22477.878} C_VEL
LIN {X 0,Y 182.735,Z 596.979,A -85,B 0,C 180,E1 -22482.079,E2 -22482.079} C_VEL
LIN {X 0,Y 179.808,Z 595.17,A -85,B 0,C 180,E1 -22486.435,E2 -22486.435} C_VEL
LIN {X 0,Y 177.445,Z 591.569,A -85,B 0,C 180,E1 -22491.977,E2 -22491.977} C_VEL
LIN {X 0,Y 176.73,Z 587.37,A -85,B 0,C 180,E1 -22496.579,E2 -22496.579} C_VEL
LIN {X 0,Y 176.457,Z 581.962,A -85,B 0,C 180,E1 -22501.139,E2 -22501.139} C_VEL
LIN {X 0,Y 176.54,Z 575.329,A -85,B 0,C 180,E1 -22505.567,E2 -22505.567} C_VEL
LIN {X 0,Y 177.054,Z 567.708,A -85,B 0,C 180,E1 -22509.71,E2 -22509.71} C_VEL
LIN {X 0,Y 177.973,Z 558.807,A -85,B 0,C 180,E1 -22513.704,E2 -22513.704} C_VEL
LIN {X 0,Y 179.227,Z 549.793,A -85,B 0,C 180,E1 -22517.101,E2 -22517.101} C_VEL
LIN {X 0,Y 180.961,Z 538.093,A -85,B 0,C 180,E1 -22520.8,E2 -22520.8} C_VEL
LIN {X 0,Y 183.064,Z 525.607,A -85,B 0,C 180,E1 -22524.071,E2 -22524.071} C_VEL
LIN {X 0,Y 185.142,Z 513.141,A -85,B 0,C 180,E1 -22526.791,E2 -22526.791} C_VEL
LIN {X 0,Y 187.622,Z 498.332,A -85,B 0,C 180,E1 -22529.446,E2 -22529.446} C_VEL
LIN {X 0,Y 189.925,Z 482.76,A -85,B 0,C 180,E1 -22531.703,E2 -22531.703} C_VEL
LIN {X 0,Y 191.954,Z 467.461,A -85,B 0,C 180,E1 -22533.466,E2 -22533.466} C_VEL
LIN {X 0,Y 193.8,Z 450.242,A -85,B 0,C 180,E1 -22534.987,E2 -22534.987} C_VEL
LIN {X 0,Y 198.546,Z 397.409,A -85,B 0,C 180,E1 -22538.274,E2 -22538.274} C_VEL
LIN {X 0,Y 202.362,Z 357.847,A -85,B 0,C 180,E1 -22540.575,E2 -22540.575} C_VEL
LIN {X 0,Y 197.406,Z 345.21,A -85,B 0,C 180,E1 -22541.993,E2 -22541.993} C_VEL
LIN {X 0,Y 186.099,Z 318.708,A -85,B 0,C 180,E1 -22545.372,E2 -22545.372} C_VEL
LIN {X 0,Y 178.448,Z 301.243,A -85,B 0,C 180,E1 -22547.871,E2 -22547.871} C_VEL
LIN {X 0,Y 178.403,Z 300.886,A -85,B 0,C 180,E1 -22547.953,E2 -22547.953} C_VEL
LIN {X 0,Y 178.436,Z 300.885,A -85,B 0,C 180,E1 -22551.97,E2 -22551.97} C_VEL
LIN {X 0,Y 178.483,Z 300.879,A -85,B 0,C 180,E1 -22556.543,E2 -22556.543} C_VEL
LIN {X 0,Y 178.442,Z 300.884,A -85,B 0,C 180,E1 -22561.792,E2 -22561.792} C_VEL
LIN {X 0,Y 178.513,Z 300.873,A -85,B 0,C 180,E1 -22564.886,E2 -22564.886} C_VEL
LIN {X 0,Y 178.587,Z 300.865,A -85,B 0,C 180,E1 -22570.812,E2 -22570.812} C_VEL
LIN {X 0,Y 178.643,Z 300.858,A -85,B 0,C 180,E1 -22576.344,E2 -22576.344} C_VEL
LIN {X 0,Y 178.955,Z 300.82,A -85,B 0,C 180,E1 -22580.959,E2 -22580.959} C_VEL
LIN {X 0,Y 179.147,Z 300.796,A -85,B 0,C 180,E1 -22587.749,E2 -22587.749} C_VEL
LIN {X 0,Y 179.364,Z 300.765,A -85,B 0,C 180,E1 -22589.997,E2 -22589.997} C_VEL
LIN {X 0,Y 178.866,Z 300.828,A -85,B 0,C 180,E1 -22594.504,E2 -22594.504} C_VEL
LIN {X 0,Y 178.956,Z 300.816,A -85,B 0,C 180,E1 -22599.035,E2 -22599.035} C_VEL
LIN {X 0,Y 178.653,Z 300.857,A -85,B 0,C 180,E1 -22603.649,E2 -22603.649} C_VEL
LIN {X 0,Y 178.614,Z 300.856,A -85,B 0,C 180,E1 -22609.214,E2 -22609.214} C_VEL
LIN {X 0,Y 178.524,Z 300.872,A -85,B 0,C 180,E1 -22615.122,E2 -22615.122} C_VEL
LIN {X 0,Y 178.466,Z 300.878,A -85,B 0,C 180,E1 -22620.789,E2 -22620.789} C_VEL
LIN {X 0,Y 178.479,Z 300.874,A -85,B 0,C 180,E1 -22624.22,E2 -22624.22} C_VEL
LIN {X 0,Y 178.406,Z 300.887,A -85,B 0,C 180,E1 -22629.067,E2 -22629.067} C_VEL
LIN {X 0,Y 178.39,Z 300.886,A -85,B 0,C 180,E1 -22632.043,E2 -22632.043} C_VEL
LIN {X 0,Y 178.382,Z 300.887,A -85,B 0,C 180,E1 -22635.163,E2 -22635.163} C_VEL
LIN {X 0,Y 178.391,Z 300.888,A -85,B 0,C 180,E1 -22638.458,E2 -22638.458} C_VEL
LIN {X 0,Y 178.41,Z 300.884,A -85,B 0,C 180,E1 -22643.783,E2 -22643.783} C_VEL
LIN {X 0,Y 178.475,Z 300.877,A -85,B 0,C 180,E1 -22646.547,E2 -22646.547} C_VEL
LIN {X 0,Y 178.511,Z 300.869,A -85,B 0,C 180,E1 -22650.006,E2 -22650.006} C_VEL
LIN {X 0,Y 178.508,Z 300.874,A -85,B 0,C 180,E1 -22654.886,E2 -22654.886} C_VEL
LIN {X 0,Y 178.609,Z 300.858,A -85,B 0,C 180,E1 -22660.787,E2 -22660.787} C_VEL
LIN {X 0,Y 178.67,Z 300.851,A -85,B 0,C 180,E1 -22666.351,E2 -22666.351} C_VEL
LIN {X 0,Y 178.948,Z 300.82,A -85,B 0,C 180,E1 -22670.963,E2 -22670.963} C_VEL
LIN {X 0,Y 179.142,Z 300.793,A -85,B 0,C 180,E1 -22677.753,E2 -22677.753} C_VEL
LIN {X 0,Y 179.359,Z 300.766,A -85,B 0,C 180,E1 -22680.002,E2 -22680.002} C_VEL
LIN {X 0,Y 178.861,Z 300.829,A -85,B 0,C 180,E1 -22684.509,E2 -22684.509} C_VEL
LIN {X 0,Y 178.95,Z 300.82,A -85,B 0,C 180,E1 -22689.04,E2 -22689.04} C_VEL
LIN {X 0,Y 178.672,Z 300.854,A -85,B 0,C 180,E1 -22693.653,E2 -22693.653} C_VEL
LIN {X 0,Y 178.613,Z 300.865,A -85,B 0,C 180,E1 -22699.217,E2 -22699.217} C_VEL
LIN {X 0,Y 178.512,Z 300.878,A -85,B 0,C 180,E1 -22705.117,E2 -22705.117} C_VEL
LIN {X 0,Y 178.494,Z 300.88,A -85,B 0,C 180,E1 -22710.789,E2 -22710.789} C_VEL
LIN {X 0,Y 178.479,Z 300.878,A -85,B 0,C 180,E1 -22714.223,E2 -22714.223} C_VEL
LIN {X 0,Y 178.482,Z 300.908,A -85,B 0,C 180,E1 -22719.327,E2 -22719.327} C_VEL
LIN {X 0,Y 179.093,Z 303.689,A -85,B 0,C 180,E1 -22720.54,E2 -22720.54} C_VEL
LIN {X 0,Y 189.576,Z 331.779,A -85,B 0,C 180,E1 -22724.222,E2 -22724.222} C_VEL
LIN {X 0,Y 202.058,Z 367.431,A -85,B 0,C 180,E1 -22728.244,E2 -22728.244} C_VEL
LIN {X 0,Y 202.783,Z 376.627,A -85,B 0,C 180,E1 -22728.943,E2 -22728.943} C_VEL
LIN {X 0,Y 194.049,Z 471.732,A -85,B 0,C 180,E1 -22734.749,E2 -22734.749} C_VEL
LIN {X 0,Y 191.975,Z 488.655,A -85,B 0,C 180,E1 -22736.224,E2 -22736.224} C_VEL
LIN {X 0,Y 190.635,Z 498.373,A -85,B 0,C 180,E1 -22737.29,E2 -22737.29} C_VEL
LIN {X 0,Y 189.82,Z 501.962,A -85,B 0,C 180,E1 -22737.709,E2 -22737.709} C_VEL
LIN {X 0,Y 187.743,Z 507.113,A -85,B 0,C 180,E1 -22738.333,E2 -22738.333} C_VEL
LIN {X 0,Y 180.835,Z 520.152,A -85,B 0,C 180,E1 -22740.207,E2 -22740.207} C_VEL
LIN {X 0,Y 179.234,Z 525.12,A -85,B 0,C 180,E1 -22741.089,E2 -22741.089} C_VEL
LIN {X 0,Y 176.761,Z 539.471,A -85,B 0,C 180,E1 -22744.068,E2 -22744.068} C_VEL
LIN {X 0,Y 174.6,Z 552.153,A -85,B 0,C 180,E1 -22747.303,E2 -22747.303} C_VEL
LIN {X 0,Y 172.799,Z 564.156,A -85,B 0,C 180,E1 -22751.016,E2 -22751.016} C_VEL
LIN {X 0,Y 171.519,Z 575.106,A -85,B 0,C 180,E1 -22755.165,E2 -22755.165} C_VEL
LIN {X 0,Y 170.84,Z 584.1,A -85,B 0,C 180,E1 -22759.335,E2 -22759.335} C_VEL
LIN {X 0,Y 170.672,Z 590.491,A -85,B 0,C 180,E1 -22762.907,E2 -22762.907} C_VEL
LIN {X 0,Y 170.666,Z 595.711,A -85,B 0,C 180,E1 -22766.462,E2 -22766.462} C_VEL
LIN {X 0,Y 170.778,Z 599.948,A -85,B 0,C 180,E1 -22770.003,E2 -22770.003} C_VEL
LIN {X 0,Y 170.399,Z 602.119,A -85,B 0,C 180,E1 -22772.367,E2 -22772.367} C_VEL
LIN {X 0,Y 169.833,Z 605.46,A -85,B 0,C 180,E1 -22777.135,E2 -22777.135} C_VEL
LIN {X 0,Y 169.898,Z 607.641,A -85,B 0,C 180,E1 -22781.94,E2 -22781.94} C_VEL
LIN {X 0,Y 171.145,Z 608.786,A -85,B 0,C 180,E1 -22786.709,E2 -22786.709} C_VEL
LIN {X 0,Y 173.72,Z 609.077,A -85,B 0,C 180,E1 -22791.486,E2 -22791.486} C_VEL
LIN {X 0,Y 179.944,Z 607.85,A -85,B 0,C 180,E1 -22797.952,E2 -22797.952} C_VEL
LIN {X 0,Y 185.523,Z 605.978,A -85,B 0,C 180,E1 -22802.032,E2 -22802.032} C_VEL
LIN {X 0,Y 192.182,Z 603.371,A -85,B 0,C 180,E1 -22805.814,E2 -22805.814} C_VEL
LIN {X 0,Y 204.424,Z 597.869,A -85,B 0,C 180,E1 -22810.787,E2 -22810.787} C_VEL
LIN {X 0,Y 216.063,Z 591.948,A -85,B 0,C 180,E1 -22814.377,E2 -22814.377} C_VEL
LIN {X 0,Y 226.208,Z 586.28,A -85,B 0,C 180,E1 -22816.88,E2 -22816.88} C_VEL
LIN {X 0,Y 216.434,Z 590.525,A -85,B 0,C 180,E1 -22819.5,E2 -22819.5} C_VEL
LIN {X 0,Y 207.429,Z 593.79,A -85,B 0,C 180,E1 -22822.419,E2 -22822.419} C_VEL
LIN {X 0,Y 199.218,Z 596.242,A -85,B 0,C 180,E1 -22825.635,E2 -22825.635} C_VEL
LIN {X 0,Y 191.706,Z 597.835,A -85,B 0,C 180,E1 -22829.118,E2 -22829.118} C_VEL
LIN {X 0,Y 185.412,Z 598.497,A -85,B 0,C 180,E1 -22832.943,E2 -22832.943} C_VEL
LIN {X 0,Y 180.102,Z 598.315,A -85,B 0,C 180,E1 -22837.03,E2 -22837.03} C_VEL
LIN {X 0,Y 175.983,Z 597.152,A -85,B 0,C 180,E1 -22841.366,E2 -22841.366} C_VEL
LIN {X 0,Y 172.903,Z 595.104,A -85,B 0,C 180,E1 -22845.882,E2 -22845.882} C_VEL
LIN {X 0,Y 170.804,Z 592.028,A -85,B 0,C 180,E1 -22850.525,E2 -22850.525} C_VEL
LIN {X 0,Y 169.811,Z 587.867,A -85,B 0,C 180,E1 -22855.25,E2 -22855.25} C_VEL
LIN {X 0,Y 169.441,Z 582.504,A -85,B 0,C 180,E1 -22859.998,E2 -22859.998} C_VEL
LIN {X 0,Y 169.441,Z 575.694,A -85,B 0,C 180,E1 -22864.757,E2 -22864.757} C_VEL
LIN {X 0,Y 169.884,Z 568.393,A -85,B 0,C 180,E1 -22868.923,E2 -22868.923} C_VEL
LIN {X 0,Y 170.716,Z 559.589,A -85,B 0,C 180,E1 -22873.085,E2 -22873.085} C_VEL
LIN {X 0,Y 172.19,Z 549.029,A -85,B 0,C 180,E1 -22877.21,E2 -22877.21} C_VEL
LIN {X 0,Y 173.952,Z 537.283,A -85,B 0,C 180,E1 -22881.01,E2 -22881.01} C_VEL
LIN {X 0,Y 175.921,Z 525.58,A -85,B 0,C 180,E1 -22884.17,E2 -22884.17} C_VEL
LIN {X 0,Y 178.054,Z 513.106,A -85,B 0,C 180,E1 -22886.993,E2 -22886.993} C_VEL
LIN {X 0,Y 180.576,Z 498.301,A -85,B 0,C 180,E1 -22889.749,E2 -22889.749} C_VEL
LIN {X 0,Y 183.023,Z 482.164,A -85,B 0,C 180,E1 -22892.16,E2 -22892.16} C_VEL
LIN {X 0,Y 185.187,Z 466.156,A -85,B 0,C 180,E1 -22894.037,E2 -22894.037} C_VEL
LIN {X 0,Y 186.996,Z 449.395,A -85,B 0,C 180,E1 -22895.545,E2 -22895.545} C_VEL
LIN {X 0,Y 195.53,Z 358.877,A -85,B 0,C 180,E1 -22901.251,E2 -22901.251} C_VEL
LIN {X 0,Y 183.951,Z 330.901,A -85,B 0,C 180,E1 -22904.73,E2 -22904.73} C_VEL
LIN {X 0,Y 172.454,Z 304.764,A -85,B 0,C 180,E1 -22908.536,E2 -22908.536} C_VEL
LIN {X 0,Y 171.338,Z 301.767,A -85,B 0,C 180,E1 -22908.979,E2 -22908.979} C_VEL
LIN {X 0,Y 171.387,Z 301.763,A -85,B 0,C 180,E1 -22912.037,E2 -22912.037} C_VEL
LIN {X 0,Y 171.397,Z 301.758,A -85,B 0,C 180,E1 -22915.089,E2 -22915.089} C_VEL
LIN {X 0,Y 171.407,Z 301.757,A -85,B 0,C 180,E1 -22920.523,E2 -22920.523} C_VEL
LIN {X 0,Y 171.438,Z 301.756,A -85,B 0,C 180,E1 -22925.795,E2 -22925.795} C_VEL
LIN {X 0,Y 171.542,Z 301.743,A -85,B 0,C 180,E1 -22930.864,E2 -22930.864} C_VEL
LIN {X 0,Y 171.557,Z 301.743,A -85,B 0,C 180,E1 -22935.768,E2 -22935.768} C_VEL
LIN {X 0,Y 171.883,Z 301.701,A -85,B 0,C 180,E1 -22940.584,E2 -22940.584} C_VEL
LIN {X 0,Y 171.815,Z 301.707,A -85,B 0,C 180,E1 -22945.304,E2 -22945.304} C_VEL
LIN {X 0,Y 172.326,Z 301.642,A -85,B 0,C 180,E1 -22949.997,E2 -22949.997} C_VEL
LIN {X 0,Y 171.815,Z 301.706,A -85,B 0,C 180,E1 -22954.689,E2 -22954.689} C_VEL
LIN {X 0,Y 171.883,Z 301.696,A -85,B 0,C 180,E1 -22959.41,E2 -22959.41} C_VEL
LIN {X 0,Y 171.57,Z 301.737,A -85,B 0,C 180,E1 -22964.224,E2 -22964.224} C_VEL
LIN {X 0,Y 171.535,Z 301.74,A -85,B 0,C 180,E1 -22969.559,E2 -22969.559} C_VEL
LIN {X 0,Y 171.458,Z 301.749,A -85,B 0,C 180,E1 -22975.614,E2 -22975.614} C_VEL
LIN {X 0,Y 171.429,Z 301.755,A -85,B 0,C 180,E1 -22980.583,E2 -22980.583} C_VEL
LIN {X 0,Y 171.39,Z 301.757,A -85,B 0,C 180,E1 -22985.031,E2 -22985.031} C_VEL
LIN {X 0,Y 171.368,Z 301.763,A -85,B 0,C 180,E1 -22988.815,E2 -22988.815} C_VEL
LIN {X 0,Y 171.31,Z 301.765,A -85,B 0,C 180,E1 -22994.216,E2 -22994.216} C_VEL
LIN {X 0,Y 171.323,Z 301.77,A -85,B 0,C 180,E1 -22998.981,E2 -22998.981} C_VEL
LIN {X 0,Y 171.374,Z 301.756,A -85,B 0,C 180,E1 -23002.04,E2 -23002.04} C_VEL
LIN {X 0,Y 171.386,Z 301.761,A -85,B 0,C 180,E1 -23005.092,E2 -23005.092} C_VEL
LIN {X 0,Y 171.437,Z 301.75,A -85,B 0,C 180,E1 -23010.534,E2 -23010.534} C_VEL
LIN {X 0,Y 171.432,Z 301.754,A -85,B 0,C 180,E1 -23015.8,E2 -23015.8} C_VEL
LIN {X 0,Y 171.565,Z 301.736,A -85,B 0,C 180,E1 -23020.872,E2 -23020.872} C_VEL
LIN {X 0,Y 171.582,Z 301.734,A -85,B 0,C 180,E1 -23025.775,E2 -23025.775} C_VEL
LIN {X 0,Y 171.877,Z 301.699,A -85,B 0,C 180,E1 -23030.588,E2 -23030.588} C_VEL
LIN {X 0,Y 171.81,Z 301.709,A -85,B 0,C 180,E1 -23035.309,E2 -23035.309} C_VEL
LIN {X 0,Y 172.322,Z 301.643,A -85,B 0,C 180,E1 -23040.002,E2 -23040.002} C_VEL
LIN {X 0,Y 171.81,Z 301.708,A -85,B 0,C 180,E1 -23044.694,E2 -23044.694} C_VEL
LIN {X 0,Y 171.879,Z 301.699,A -85,B 0,C 180,E1 -23049.415,E2 -23049.415} C_VEL
LIN {X 0,Y 171.585,Z 301.737,A -85,B 0,C 180,E1 -23054.228,E2 -23054.228} C_VEL
LIN {X 0,Y 171.532,Z 301.746,A -85,B 0,C 180,E1 -23059.56,E2 -23059.56} C_VEL
LIN {X 0,Y 171.451,Z 301.756,A -85,B 0,C 180,E1 -23065.612,E2 -23065.612} C_VEL
LIN {X 0,Y 171.452,Z 301.756,A -85,B 0,C 180,E1 -23070.599,E2 -23070.599} C_VEL
LIN {X 0,Y 171.387,Z 301.762,A -85,B 0,C 180,E1 -23075.038,E2 -23075.038} C_VEL
LIN {X 0,Y 171.442,Z 301.771,A -85,B 0,C 180,E1 -23078.643,E2 -23078.643} C_VEL
LIN {X 0,Y 171.789,Z 303.409,A -85,B 0,C 180,E1 -23079.331,E2 -23079.331} C_VEL
LIN {X 0,Y 182.756,Z 332.932,A -85,B 0,C 180,E1 -23083.39,E2 -23083.39} C_VEL
LIN {X 0,Y 194.357,Z 365.966,A -85,B 0,C 180,E1 -23087.297,E2 -23087.297} C_VEL
LIN {X 0,Y 195.633,Z 370.64,A -85,B 0,C 180,E1 -23087.769,E2 -23087.769} C_VEL
LIN {X 0,Y 196.076,Z 377.025,A -85,B 0,C 180,E1 -23088.266,E2 -23088.266} C_VEL
LIN {X 0,Y 187.107,Z 471.813,A -85,B 0,C 180,E1 -23094.316,E2 -23094.316} C_VEL
LIN {X 0,Y 184.945,Z 489.107,A -85,B 0,C 180,E1 -23095.913,E2 -23095.913} C_VEL
LIN {X 0,Y 182.534,Z 505.331,A -85,B 0,C 180,E1 -23097.895,E2 -23097.895} C_VEL
LIN {X 0,Y 180.121,Z 520.019,A -85,B 0,C 180,E1 -23100.17,E2 -23100.17} C_VEL
LIN {X 0,Y 179.234,Z 525.12,A -85,B 0,C 180,E1 -23101.089,E2 -23101.089} C_VEL
LIN {X 0,Y 177.647,Z 530.04,A -85,B 0,C 180,E1 -23102.026,E2 -23102.026} C_VEL
LIN {X 0,Y 173.418,Z 537.528,A -85,B 0,C 180,E1 -23103.633,E2 -23103.633} C_VEL
LIN {X 0,Y 169.294,Z 544.767,A -85,B 0,C 180,E1 -23105.449,E2 -23105.449} C_VEL
LIN {X 0,Y 167.894,Z 549.217,A -85,B 0,C 180,E1 -23106.688,E2 -23106.688} C_VEL
LIN {X 0,Y 166.165,Z 560.617,A -85,B 0,C 180,E1 -23110.227,E2 -23110.227} C_VEL
LIN {X 0,Y 164.723,Z 572.062,A -85,B 0,C 180,E1 -23114.538,E2 -23114.538} C_VEL
LIN {X 0,Y 163.959,Z 581.47,A -85,B 0,C 180,E1 -23118.882,E2 -23118.882} C_VEL
LIN {X 0,Y 163.784,Z 589.159,A -85,B 0,C 180,E1 -23123.227,E2 -23123.227} C_VEL
LIN {X 0,Y 163.77,Z 593.684,A -85,B 0,C 180,E1 -23126.313,E2 -23126.313} C_VEL
LIN {X 0,Y 163.871,Z 598.122,A -85,B 0,C 180,E1 -23130.003,E2 -23130.003} C_VEL
LIN {X 0,Y 163.502,Z 600.451,A -85,B 0,C 180,E1 -23132.467,E2 -23132.467} C_VEL
LIN {X 0,Y 162.912,Z 604.018,A -85,B 0,C 180,E1 -23137.439,E2 -23137.439} C_VEL
LIN {X 0,Y 163.009,Z 606.388,A -85,B 0,C 180,E1 -23142.452,E2 -23142.452} C_VEL
LIN {X 0,Y 164.34,Z 607.838,A -85,B 0,C 180,E1 -23147.422,E2 -23147.422} C_VEL
LIN {X 0,Y 167.021,Z 608.335,A -85,B 0,C 180,E1 -23152.257,E2 -23152.257} C_VEL
LIN {X 0,Y 171.158,Z 608.054,A -85,B 0,C 180,E1 -23156.855,E2 -23156.855} C_VEL
LIN {X 0,Y 179.515,Z 606.075,A -85,B 0,C 180,E1 -23163.24,E2 -23163.24} C_VEL
LIN {X 0,Y 186.481,Z 603.752,A -85,B 0,C 180,E1 -23167.088,E2 -23167.088} C_VEL
LIN {X 0,Y 194.711,Z 600.712,A -85,B 0,C 180,E1 -23170.522,E2 -23170.522} C_VEL
LIN {X 0,Y 206.222,Z 595.786,A -85,B 0,C 180,E1 -23174.321,E2 -23174.321} C_VEL
LIN {X 0,Y 216.302,Z 591.023,A -85,B 0,C 180,E1 -23176.973,E2 -23176.973} C_VEL
LIN {X 0,Y 206.613,Z 594.307,A -85,B 0,C 180,E1 -23179.736,E2 -23179.736} C_VEL
LIN {X 0,Y 197.692,Z 596.804,A -85,B 0,C 180,E1 -23182.816,E2 -23182.816} C_VEL
LIN {X 0,Y 185.74,Z 598.912,A -85,B 0,C 180,E1 -23188.011,E2 -23188.011} C_VEL
LIN {X 0,Y 179.168,Z 599.26,A -85,B 0,C 180,E1 -23191.918,E2 -23191.918} C_VEL
LIN {X 0,Y 173.609,Z 598.693,A -85,B 0,C 180,E1 -23196.119,E2 -23196.119} C_VEL
LIN {X 0,Y 169.271,Z 597.287,A -85,B 0,C 180,E1 -23200.599,E2 -23200.599} C_VEL
LIN {X 0,Y 166.026,Z 594.887,A -85,B 0,C 180,E1 -23205.285,E2 -23205.285} C_VEL
LIN {X 0,Y 163.826,Z 591.528,A -85,B 0,C 180,E1 -23210.117,E2 -23210.117} C_VEL
LIN {X 0,Y 162.774,Z 587.127,A -85,B 0,C 180,E1 -23215.044,E2 -23215.044} C_VEL
LIN {X 0,Y 162.458,Z 582.978,A -85,B 0,C 180,E1 -23218.759,E2 -23218.759} C_VEL
LIN {X 0,Y 162.365,Z 576.834,A -85,B 0,C 180,E1 -23223.33,E2 -23223.33} C_VEL
